// TIA Portal V20 export
FUNCTION_BLOCK "Sequence_10_GaugeRnR"   // FB244, LAD
AUTHOR : ERsystem_FA2_DH. Kim
// stored: IsIECCheckEnabled true, MemoryReserve 100, Namespace Unit1.Em5, SetENOAutomatically false
   VAR_INPUT
      unitStatus : "LAF_typeUnitStatus";
   END_VAR
   VAR
      statSelectedJobNumber { ExternalWritable := 'False'} : DInt;   // Evaluated Job Number
      instSequenceLADStatus { ExternalWritable := 'False'} : "LAF_StatusLadSequence";
      instSequenceLADControl { ExternalWritable := 'False'} : "LAF_ControlLadSequence";
   END_VAR
   VAR CONSTANT
      STEP_IDLE : DInt := 1;
      STEP_IMMEDIATE_STOP : DInt := 9001;   // Step executed when an immediate stop command is triggered for the sequence (i.e. when unit is in state aborting)
      JOB_1_STEP_01 : DInt := 101;
      JOB_1_STEP_10 : DInt := 110;
      JOB_1_STEP_20 : DInt := 120;
      JOB_1_STEP_30 : DInt := 130;
      JOB_1_STEP_90 : DInt := 190;
      JOB_2_STEP_01 : DInt := 201;
      JOB_2_STEP_10 : DInt := 210;
      JOB_2_STEP_20 : DInt := 220;
      JOB_2_STEP_30 : DInt := 230;
      JOB_2_STEP_40 : DInt := 240;
      JOB_2_STEP_50 : DInt := 250;
      JOB_2_STEP_90 : DInt := 290;
      JOB_3_STEP_01 : DInt := 301;
      JOB_3_STEP_10 : DInt := 310;
      JOB_3_STEP_20 : DInt := 320;
      JOB_3_STEP_90 : DInt := 390;
      JOB_4_STEP_01 : DInt := 401;
      JOB_4_STEP_10 : DInt := 410;
      JOB_4_STEP_20 : DInt := 420;
      JOB_4_STEP_30 : DInt := 430;
      JOB_4_STEP_40 : DInt := 440;
      JOB_4_STEP_90 : DInt := 490;
      JOB_5_STEP_01 : DInt := 501;
      JOB_5_STEP_10 : DInt := 510;
      JOB_5_STEP_20 : DInt := 520;
      JOB_5_STEP_90 : DInt := 590;
      JOB_6_STEP_01 : DInt := 601;
      JOB_6_STEP_10 : DInt := 610;
      JOB_6_STEP_20 : DInt := 620;
      JOB_6_STEP_90 : DInt := 690;
      JOB_10_STEP_01 : DInt := 1001;
      JOB_10_STEP_10 : DInt := 1010;
      JOB_10_STEP_20 : DInt := 1020;
      JOB_10_STEP_30 : DInt := 1030;
      JOB_10_STEP_40 : DInt := 1040;
      JOB_10_STEP_90 : DInt := 1090;
      JOB_11_STEP_01 : DInt := 1101;
      JOB_11_STEP_10 : DInt := 1110;
      JOB_11_STEP_20 : DInt := 1120;
      JOB_11_STEP_90 : DInt := 1190;
      JOB_12_STEP_01 : DInt := 1201;
      JOB_12_STEP_10 : DInt := 1210;
      JOB_12_STEP_90 : DInt := 1290;
      JOB_13_STEP_01 : DInt := 1301;
      JOB_13_STEP_10 : DInt := 1310;
      JOB_13_STEP_20 : DInt := 1320;
      JOB_13_STEP_30 : DInt := 1330;
      JOB_13_STEP_40 : DInt := 1340;
      JOB_13_STEP_50 : DInt := 1350;
      JOB_13_STEP_90 : DInt := 1390;
      JOB_15_STEP_01 : DInt := 1501;
      JOB_15_STEP_10 : DInt := 1510;
      JOB_15_STEP_20 : DInt := 1520;
      JOB_15_STEP_90 : DInt := 1590;
      JOB_16_STEP_01 : DInt := 1601;
      JOB_16_STEP_10 : DInt := 1610;
      JOB_16_STEP_20 : DInt := 1620;
      JOB_16_STEP_30 : DInt := 1630;
      JOB_16_STEP_40 : DInt := 1640;
      JOB_16_STEP_90 : DInt := 1690;
      JOB_17_STEP_01 : DInt := 1701;
      JOB_17_STEP_10 : DInt := 1710;
      JOB_17_STEP_20 : DInt := 1720;
      JOB_17_STEP_90 : DInt := 1790;
      JOB_18_STEP_01 : DInt := 1801;
      JOB_18_STEP_10 : DInt := 1810;
      JOB_18_STEP_90 : DInt := 1890;
      JOB_19_STEP_01 : DInt := 1901;
      JOB_19_STEP_10 : DInt := 1910;
      JOB_19_STEP_20 : DInt := 1920;
      JOB_19_STEP_30 : DInt := 1930;
      JOB_19_STEP_40 : DInt := 1940;
      JOB_19_STEP_90 : DInt := 1990;
      JOB_20_STEP_01 : DInt := 2001;
      JOB_20_STEP_10 : DInt := 2010;
      JOB_20_STEP_20 : DInt := 2020;
      JOB_20_STEP_30 : DInt := 2030;
      JOB_20_STEP_40 : DInt := 2040;
      JOB_20_STEP_90 : DInt := 2090;
      JOB_21_STEP_01 : DInt := 2101;
      JOB_21_STEP_10 : DInt := 2110;
      JOB_21_STEP_20 : DInt := 2120;
      JOB_21_STEP_90 : DInt := 2190;
      JOB_22_STEP_01 : DInt := 2201;
      JOB_22_STEP_10 : DInt := 2210;
      JOB_22_STEP_20 : DInt := 2220;
      JOB_22_STEP_30 : DInt := 2230;
      JOB_22_STEP_40 : DInt := 2240;
      JOB_22_STEP_90 : DInt := 2290;
      JOB_23_STEP_01 : DInt := 2301;
      JOB_23_STEP_10 : DInt := 2310;
      JOB_23_STEP_20 : DInt := 2320;
      JOB_23_STEP_90 : DInt := 2390;
      JOB_24_STEP_01 : DInt := 2401;
      JOB_24_STEP_10 : DInt := 2410;
      JOB_24_STEP_20 : DInt := 2420;
      JOB_24_STEP_30 : DInt := 2430;
      JOB_24_STEP_40 : DInt := 2440;
      JOB_24_STEP_90 : DInt := 2490;
      JOB_25_STEP_01 : DInt := 2501;
      JOB_25_STEP_10 : DInt := 2510;
      JOB_25_STEP_20 : DInt := 2520;
      JOB_25_STEP_90 : DInt := 2590;
      JOB_26_STEP_01 : DInt := 2601;
      JOB_26_STEP_10 : DInt := 2610;
      JOB_26_STEP_20 : DInt := 2620;
      JOB_26_STEP_30 : DInt := 2630;
      JOB_26_STEP_40 : DInt := 2640;
      JOB_26_STEP_50 : DInt := 2650;
      JOB_26_STEP_90 : DInt := 2690;
      JOB_30_STEP_01 : DInt := 3001;
      JOB_30_STEP_10 : DInt := 3010;
      JOB_30_STEP_90 : DInt := 3090;
      JOB_31_STEP_01 : DInt := 3101;
      JOB_31_STEP_10 : DInt := 3110;
      JOB_31_STEP_15 : DInt := 3115;
      JOB_31_STEP_20 : DInt := 3120;
      JOB_31_STEP_25 : DInt := 3125;
      JOB_31_STEP_30 : DInt := 3130;
      JOB_31_STEP_35 : DInt := 3135;
      JOB_31_STEP_40 : DInt := 3140;
      JOB_31_STEP_45 : DInt := 3145;
      JOB_31_STEP_50 : DInt := 3150;
      JOB_31_STEP_55 : DInt := 3155;
      JOB_31_STEP_60 : DInt := 3160;
      JOB_31_STEP_65 : DInt := 3165;
      JOB_31_STEP_70 : DInt := 3170;
      JOB_31_STEP_90 : DInt := 3190;
      JOB_32_STEP_01 : DInt := 3201;
      JOB_32_STEP_10 : DInt := 3210;
      JOB_32_STEP_20 : DInt := 3220;
      JOB_32_STEP_90 : DInt := 3290;
      JOB_33_STEP_01 : DInt := 3301;
      JOB_33_STEP_10 : DInt := 3310;
      JOB_33_STEP_90 : DInt := 3390;
      JOB_39_STEP_01 : DInt := 3901;
      JOB_39_STEP_10 : DInt := 3910;
      JOB_39_STEP_90 : DInt := 3990;
   END_VAR
   VAR_TEMP   // added for the SCL form of the ladder/FBD networks
      _w1 : Bool;
   END_VAR
BEGIN

REGION Network 1: BLOCK INFO HEADER
   // (company) / (C) Copyright (year)
   // ---------------------------------------------------------------------------------
   // Title:                             (Title of this block)
   // Comment/Function: (that is implemented in the block)
   // Library/Family:           (that the source is dedicated to)
   // Author:                        (department / person in charge / contact)
   // Target System:          (test system with FW version)
   // Engineering:              TIA Portal (SW version)
   // Restrictions:               (OB types, etc.)
   // Requirements:           (hardware, technological package, etc.)
   // ---------------------------------------------------------------------------------
   // Change log table:
   // Version          | Date             | Signature      | Expert in charge  | Changes applied ------------------------|----------------------|-------------------------|--------------------------------|-----------------------
   // 001.000.000 | yyyy-mm-dd | 0x00000000 | (name of expert) | First released version
END_REGION

REGION Network 2: DESCRIPTION
   // This is a template block provided by the Automation Framework. It can be used to create an own project.
   // The Block Info Header is prepared to put in your own data.
   // Description of the block could be added here and the docu created by Code2Docu.
END_REGION

REGION Network 3: ********************* CONTROL *************************
END_REGION

REGION Network 4: Sequence Control
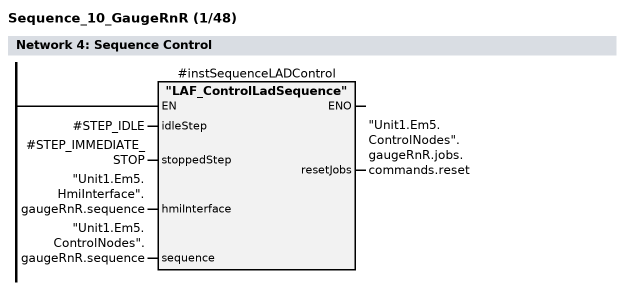
   RUNG wire#powerrail
      #instSequenceLADControl(idleStep := #STEP_IDLE, stoppedStep := #STEP_IMMEDIATE_STOP, hmiInterface := "Unit1.Em5.HmiInterface".gaugeRnR.sequence, sequence := "Unit1.Em5.ControlNodes".gaugeRnR.sequence, resetJobs => "Unit1.Em5.ControlNodes".gaugeRnR.jobs.commands.reset)
   END_RUNG
   // the same network as SCL:
   #instSequenceLADControl(idleStep := #STEP_IDLE,   // "LAF_ControlLadSequence"
                           stoppedStep := #STEP_IMMEDIATE_STOP,
                           hmiInterface := "Unit1.Em5.HmiInterface".gaugeRnR.sequence,
                           sequence := "Unit1.Em5.ControlNodes".gaugeRnR.sequence,
                           resetJobs => "Unit1.Em5.ControlNodes".gaugeRnR.jobs.commands.reset);
END_REGION

REGION Network 5: *************** JOB SELECT **************************
END_REGION

REGION Network 6: STEP IDLE
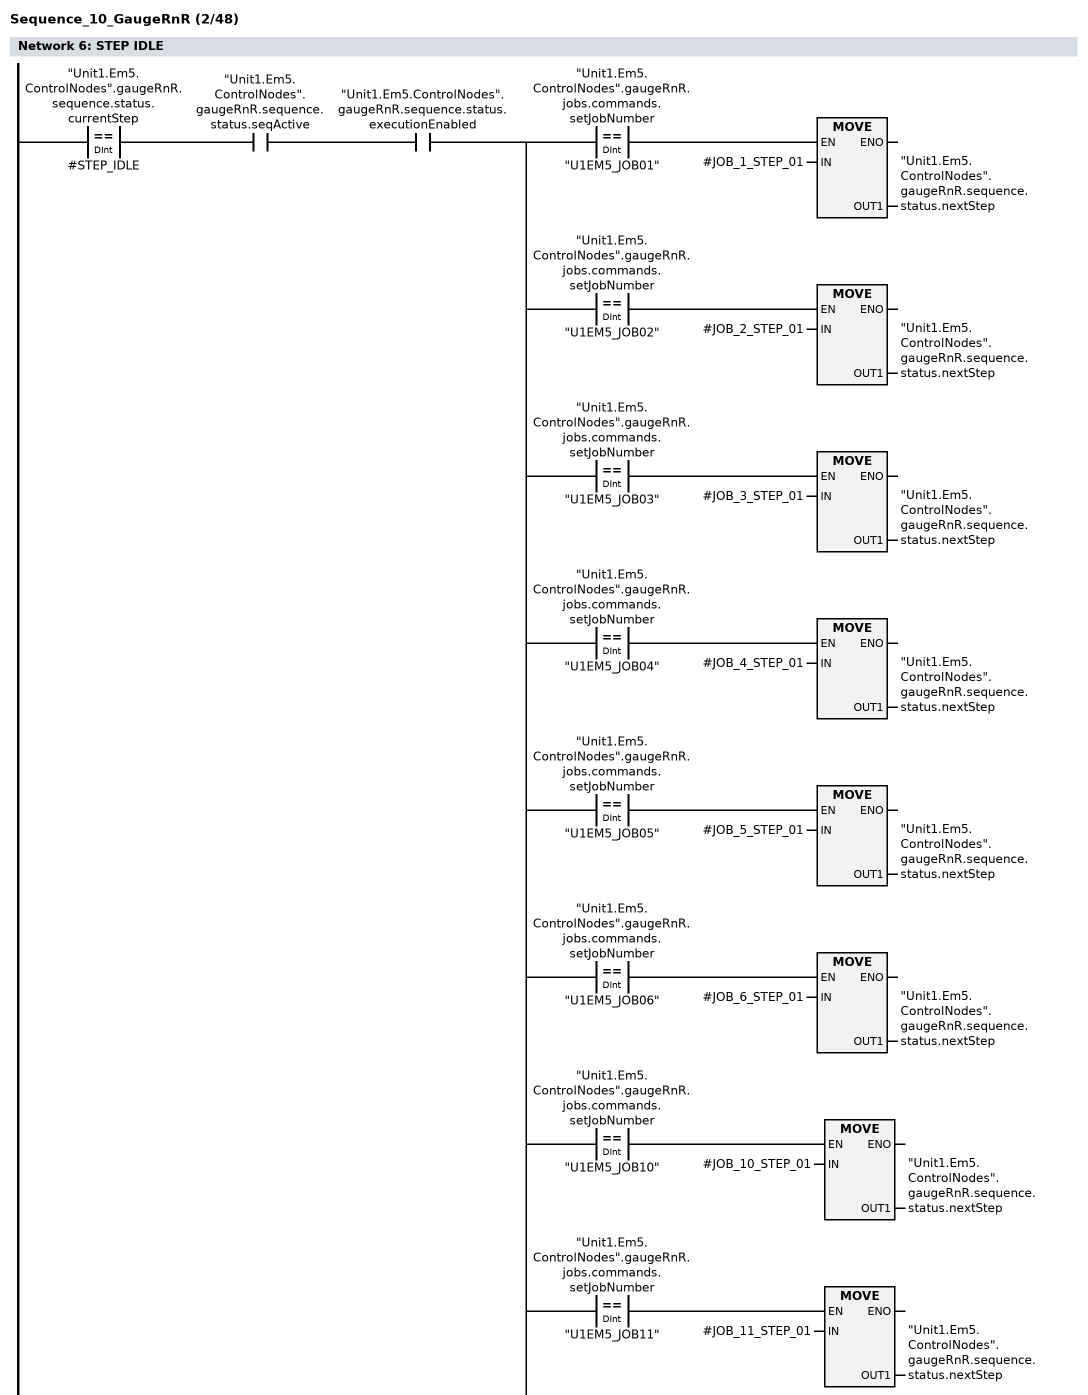
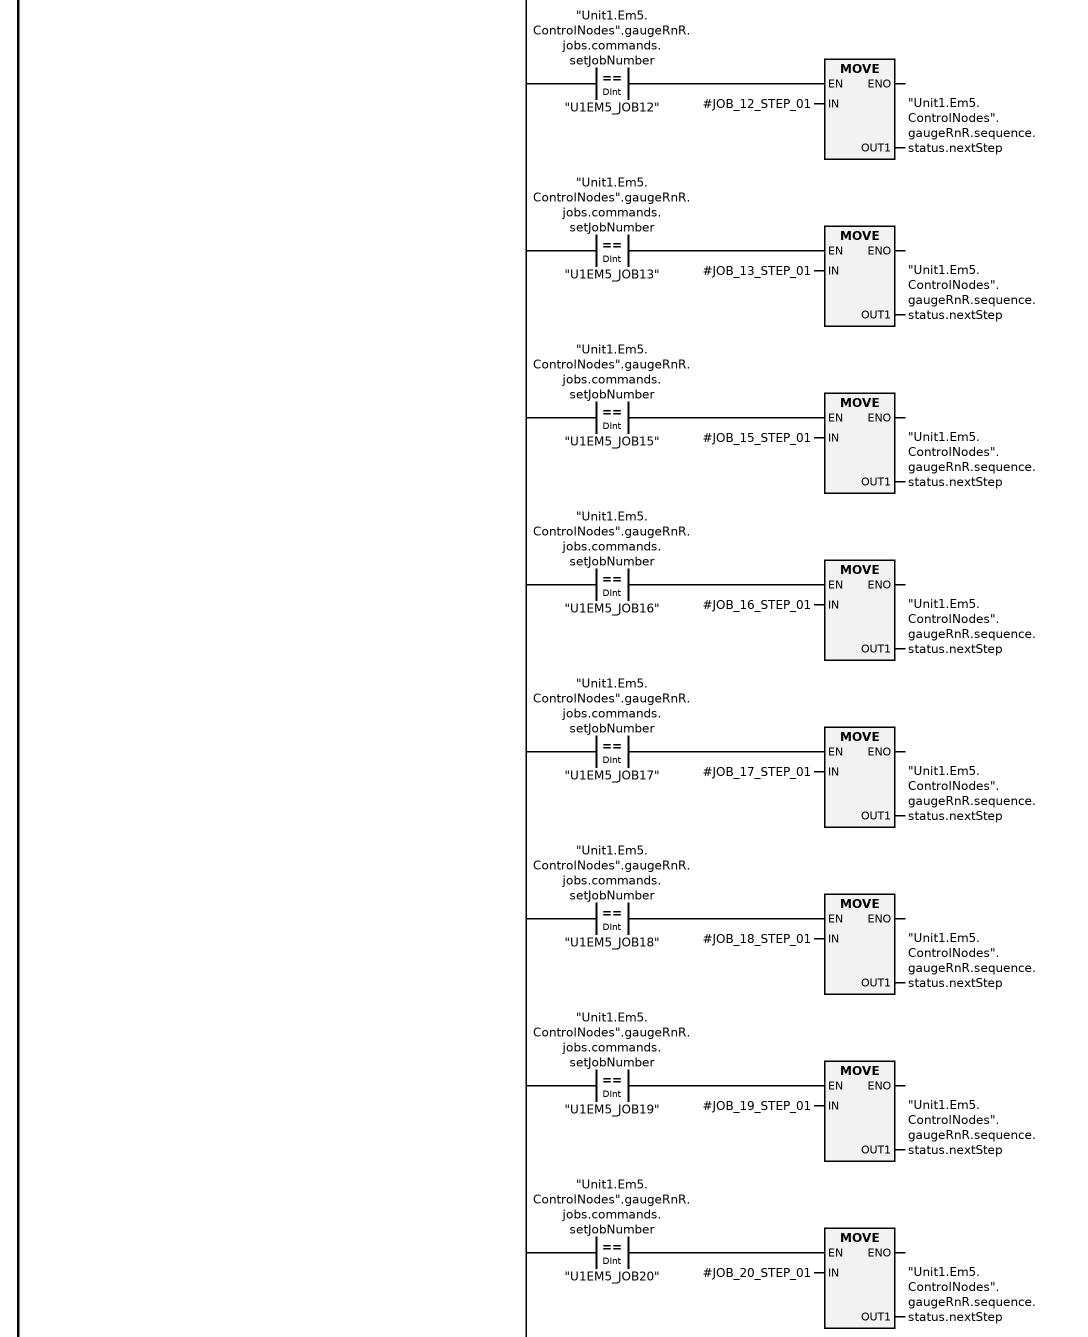
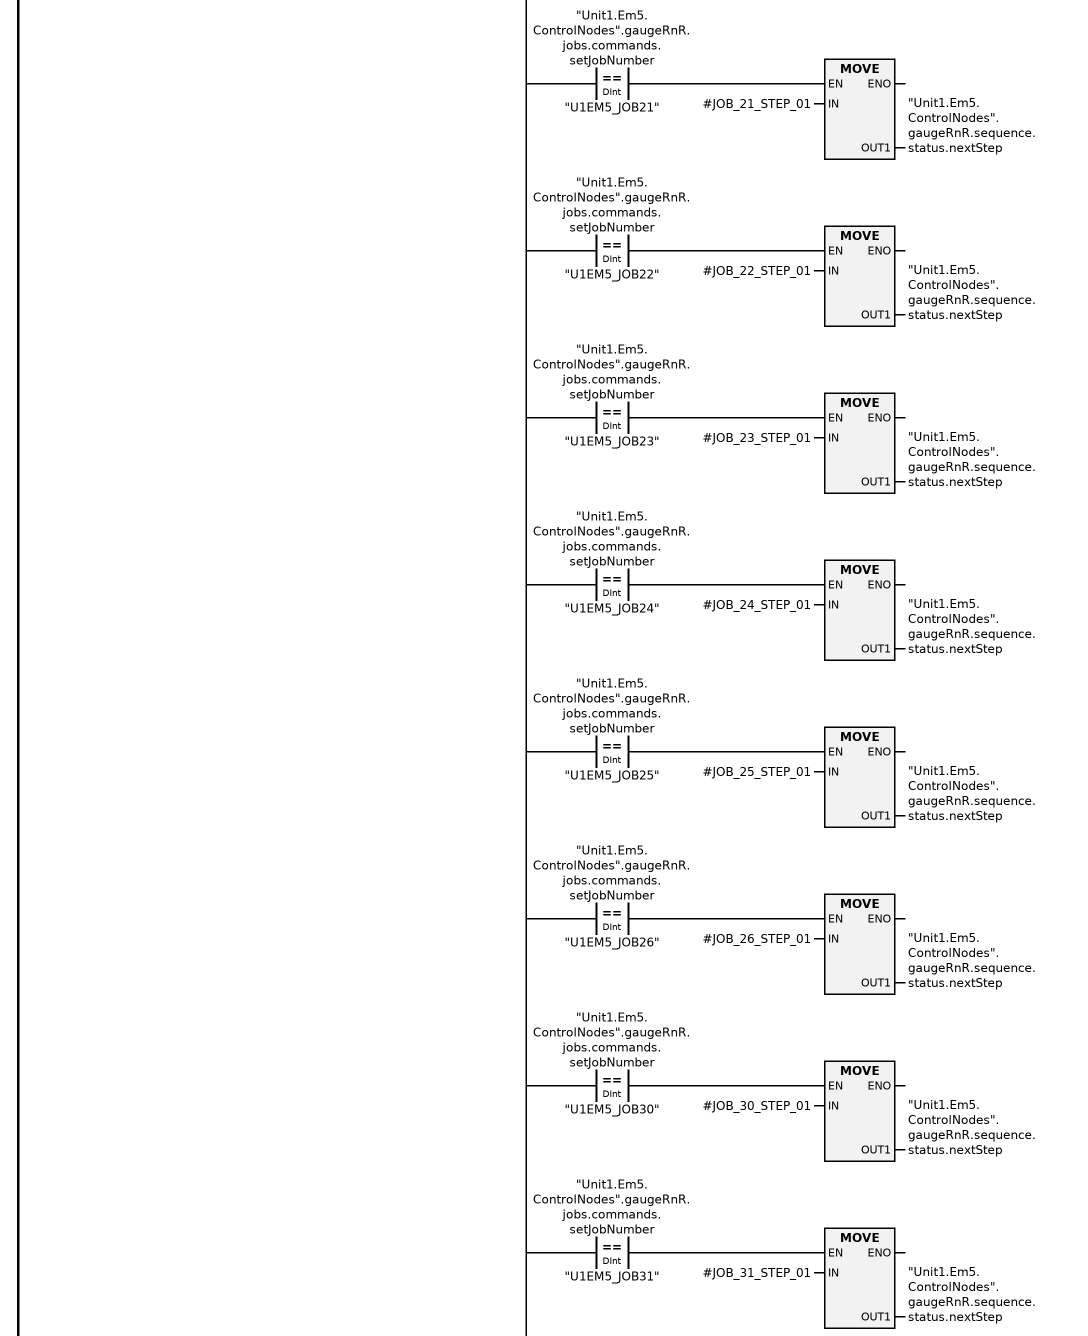
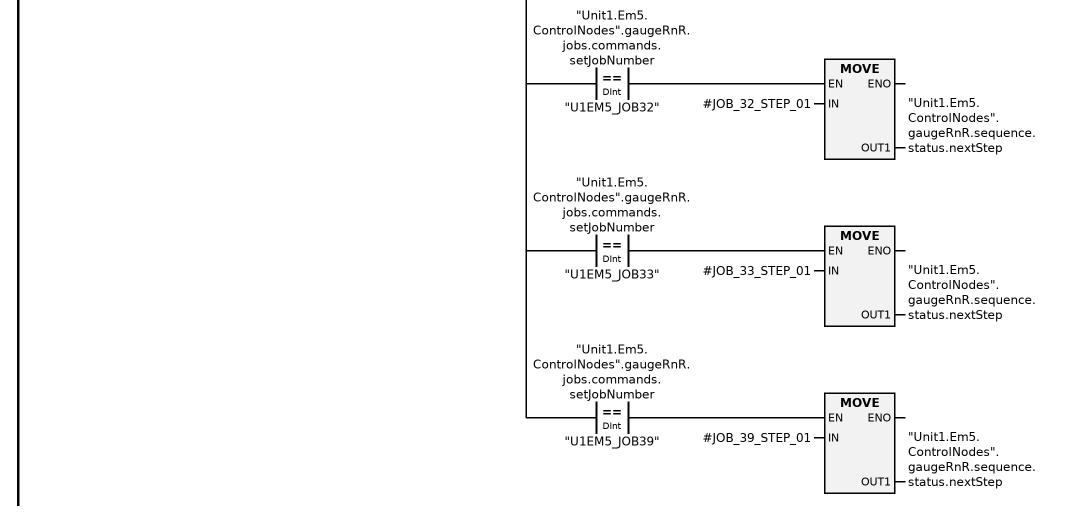
   RUNG wire#powerrail
      { S7_Templates := "SrcType := DInt" } EQ_Contact(in1 := "Unit1.Em5.ControlNodes".gaugeRnR.sequence.status.currentStep, in2 := #STEP_IDLE)
      Contact( "Unit1.Em5.ControlNodes".gaugeRnR.sequence.status.seqActive )
      Contact( "Unit1.Em5.ControlNodes".gaugeRnR.sequence.status.executionEnabled )
      wire#w1
      { S7_Templates := "SrcType := DInt" } EQ_Contact(in1 := "Unit1.Em5.ControlNodes".gaugeRnR.jobs.commands.setJobNumber, in2 := "U1EM5_JOB01")
      Move(in := #JOB_1_STEP_01, out1 => "Unit1.Em5.ControlNodes".gaugeRnR.sequence.status.nextStep)
   END_RUNG
   RUNG wire#w1
      { S7_Templates := "SrcType := DInt" } EQ_Contact(in1 := "Unit1.Em5.ControlNodes".gaugeRnR.jobs.commands.setJobNumber, in2 := "U1EM5_JOB02")
      Move(in := #JOB_2_STEP_01, out1 => "Unit1.Em5.ControlNodes".gaugeRnR.sequence.status.nextStep)
   END_RUNG
   RUNG wire#w1
      { S7_Templates := "SrcType := DInt" } EQ_Contact(in1 := "Unit1.Em5.ControlNodes".gaugeRnR.jobs.commands.setJobNumber, in2 := "U1EM5_JOB03")
      Move(in := #JOB_3_STEP_01, out1 => "Unit1.Em5.ControlNodes".gaugeRnR.sequence.status.nextStep)
   END_RUNG
   RUNG wire#w1
      { S7_Templates := "SrcType := DInt" } EQ_Contact(in1 := "Unit1.Em5.ControlNodes".gaugeRnR.jobs.commands.setJobNumber, in2 := "U1EM5_JOB04")
      Move(in := #JOB_4_STEP_01, out1 => "Unit1.Em5.ControlNodes".gaugeRnR.sequence.status.nextStep)
   END_RUNG
   RUNG wire#w1
      { S7_Templates := "SrcType := DInt" } EQ_Contact(in1 := "Unit1.Em5.ControlNodes".gaugeRnR.jobs.commands.setJobNumber, in2 := "U1EM5_JOB05")
      Move(in := #JOB_5_STEP_01, out1 => "Unit1.Em5.ControlNodes".gaugeRnR.sequence.status.nextStep)
   END_RUNG
   RUNG wire#w1
      { S7_Templates := "SrcType := DInt" } EQ_Contact(in1 := "Unit1.Em5.ControlNodes".gaugeRnR.jobs.commands.setJobNumber, in2 := "U1EM5_JOB06")
      Move(in := #JOB_6_STEP_01, out1 => "Unit1.Em5.ControlNodes".gaugeRnR.sequence.status.nextStep)
   END_RUNG
   RUNG wire#w1
      { S7_Templates := "SrcType := DInt" } EQ_Contact(in1 := "Unit1.Em5.ControlNodes".gaugeRnR.jobs.commands.setJobNumber, in2 := "U1EM5_JOB10")
      Move(in := #JOB_10_STEP_01, out1 => "Unit1.Em5.ControlNodes".gaugeRnR.sequence.status.nextStep)
   END_RUNG
   RUNG wire#w1
      { S7_Templates := "SrcType := DInt" } EQ_Contact(in1 := "Unit1.Em5.ControlNodes".gaugeRnR.jobs.commands.setJobNumber, in2 := "U1EM5_JOB11")
      Move(in := #JOB_11_STEP_01, out1 => "Unit1.Em5.ControlNodes".gaugeRnR.sequence.status.nextStep)
   END_RUNG
   RUNG wire#w1
      { S7_Templates := "SrcType := DInt" } EQ_Contact(in1 := "Unit1.Em5.ControlNodes".gaugeRnR.jobs.commands.setJobNumber, in2 := "U1EM5_JOB12")
      Move(in := #JOB_12_STEP_01, out1 => "Unit1.Em5.ControlNodes".gaugeRnR.sequence.status.nextStep)
   END_RUNG
   RUNG wire#w1
      { S7_Templates := "SrcType := DInt" } EQ_Contact(in1 := "Unit1.Em5.ControlNodes".gaugeRnR.jobs.commands.setJobNumber, in2 := "U1EM5_JOB13")
      Move(in := #JOB_13_STEP_01, out1 => "Unit1.Em5.ControlNodes".gaugeRnR.sequence.status.nextStep)
   END_RUNG
   RUNG wire#w1
      { S7_Templates := "SrcType := DInt" } EQ_Contact(in1 := "Unit1.Em5.ControlNodes".gaugeRnR.jobs.commands.setJobNumber, in2 := "U1EM5_JOB15")
      Move(in := #JOB_15_STEP_01, out1 => "Unit1.Em5.ControlNodes".gaugeRnR.sequence.status.nextStep)
   END_RUNG
   RUNG wire#w1
      { S7_Templates := "SrcType := DInt" } EQ_Contact(in1 := "Unit1.Em5.ControlNodes".gaugeRnR.jobs.commands.setJobNumber, in2 := "U1EM5_JOB16")
      Move(in := #JOB_16_STEP_01, out1 => "Unit1.Em5.ControlNodes".gaugeRnR.sequence.status.nextStep)
   END_RUNG
   RUNG wire#w1
      { S7_Templates := "SrcType := DInt" } EQ_Contact(in1 := "Unit1.Em5.ControlNodes".gaugeRnR.jobs.commands.setJobNumber, in2 := "U1EM5_JOB17")
      Move(in := #JOB_17_STEP_01, out1 => "Unit1.Em5.ControlNodes".gaugeRnR.sequence.status.nextStep)
   END_RUNG
   RUNG wire#w1
      { S7_Templates := "SrcType := DInt" } EQ_Contact(in1 := "Unit1.Em5.ControlNodes".gaugeRnR.jobs.commands.setJobNumber, in2 := "U1EM5_JOB18")
      Move(in := #JOB_18_STEP_01, out1 => "Unit1.Em5.ControlNodes".gaugeRnR.sequence.status.nextStep)
   END_RUNG
   RUNG wire#w1
      { S7_Templates := "SrcType := DInt" } EQ_Contact(in1 := "Unit1.Em5.ControlNodes".gaugeRnR.jobs.commands.setJobNumber, in2 := "U1EM5_JOB19")
      Move(in := #JOB_19_STEP_01, out1 => "Unit1.Em5.ControlNodes".gaugeRnR.sequence.status.nextStep)
   END_RUNG
   RUNG wire#w1
      { S7_Templates := "SrcType := DInt" } EQ_Contact(in1 := "Unit1.Em5.ControlNodes".gaugeRnR.jobs.commands.setJobNumber, in2 := "U1EM5_JOB20")
      Move(in := #JOB_20_STEP_01, out1 => "Unit1.Em5.ControlNodes".gaugeRnR.sequence.status.nextStep)
   END_RUNG
   RUNG wire#w1
      { S7_Templates := "SrcType := DInt" } EQ_Contact(in1 := "Unit1.Em5.ControlNodes".gaugeRnR.jobs.commands.setJobNumber, in2 := "U1EM5_JOB21")
      Move(in := #JOB_21_STEP_01, out1 => "Unit1.Em5.ControlNodes".gaugeRnR.sequence.status.nextStep)
   END_RUNG
   RUNG wire#w1
      { S7_Templates := "SrcType := DInt" } EQ_Contact(in1 := "Unit1.Em5.ControlNodes".gaugeRnR.jobs.commands.setJobNumber, in2 := "U1EM5_JOB22")
      Move(in := #JOB_22_STEP_01, out1 => "Unit1.Em5.ControlNodes".gaugeRnR.sequence.status.nextStep)
   END_RUNG
   RUNG wire#w1
      { S7_Templates := "SrcType := DInt" } EQ_Contact(in1 := "Unit1.Em5.ControlNodes".gaugeRnR.jobs.commands.setJobNumber, in2 := "U1EM5_JOB23")
      Move(in := #JOB_23_STEP_01, out1 => "Unit1.Em5.ControlNodes".gaugeRnR.sequence.status.nextStep)
   END_RUNG
   RUNG wire#w1
      { S7_Templates := "SrcType := DInt" } EQ_Contact(in1 := "Unit1.Em5.ControlNodes".gaugeRnR.jobs.commands.setJobNumber, in2 := "U1EM5_JOB24")
      Move(in := #JOB_24_STEP_01, out1 => "Unit1.Em5.ControlNodes".gaugeRnR.sequence.status.nextStep)
   END_RUNG
   RUNG wire#w1
      { S7_Templates := "SrcType := DInt" } EQ_Contact(in1 := "Unit1.Em5.ControlNodes".gaugeRnR.jobs.commands.setJobNumber, in2 := "U1EM5_JOB25")
      Move(in := #JOB_25_STEP_01, out1 => "Unit1.Em5.ControlNodes".gaugeRnR.sequence.status.nextStep)
   END_RUNG
   RUNG wire#w1
      { S7_Templates := "SrcType := DInt" } EQ_Contact(in1 := "Unit1.Em5.ControlNodes".gaugeRnR.jobs.commands.setJobNumber, in2 := "U1EM5_JOB26")
      Move(in := #JOB_26_STEP_01, out1 => "Unit1.Em5.ControlNodes".gaugeRnR.sequence.status.nextStep)
   END_RUNG
   RUNG wire#w1
      { S7_Templates := "SrcType := DInt" } EQ_Contact(in1 := "Unit1.Em5.ControlNodes".gaugeRnR.jobs.commands.setJobNumber, in2 := "U1EM5_JOB30")
      Move(in := #JOB_30_STEP_01, out1 => "Unit1.Em5.ControlNodes".gaugeRnR.sequence.status.nextStep)
   END_RUNG
   RUNG wire#w1
      { S7_Templates := "SrcType := DInt" } EQ_Contact(in1 := "Unit1.Em5.ControlNodes".gaugeRnR.jobs.commands.setJobNumber, in2 := "U1EM5_JOB31")
      Move(in := #JOB_31_STEP_01, out1 => "Unit1.Em5.ControlNodes".gaugeRnR.sequence.status.nextStep)
   END_RUNG
   RUNG wire#w1
      { S7_Templates := "SrcType := DInt" } EQ_Contact(in1 := "Unit1.Em5.ControlNodes".gaugeRnR.jobs.commands.setJobNumber, in2 := "U1EM5_JOB32")
      Move(in := #JOB_32_STEP_01, out1 => "Unit1.Em5.ControlNodes".gaugeRnR.sequence.status.nextStep)
   END_RUNG
   RUNG wire#w1
      { S7_Templates := "SrcType := DInt" } EQ_Contact(in1 := "Unit1.Em5.ControlNodes".gaugeRnR.jobs.commands.setJobNumber, in2 := "U1EM5_JOB33")
      Move(in := #JOB_33_STEP_01, out1 => "Unit1.Em5.ControlNodes".gaugeRnR.sequence.status.nextStep)
   END_RUNG
   RUNG wire#w1
      { S7_Templates := "SrcType := DInt" } EQ_Contact(in1 := "Unit1.Em5.ControlNodes".gaugeRnR.jobs.commands.setJobNumber, in2 := "U1EM5_JOB39")
      Move(in := #JOB_39_STEP_01, out1 => "Unit1.Em5.ControlNodes".gaugeRnR.sequence.status.nextStep)
   END_RUNG
   // the same network as SCL:
   #_w1 := ("Unit1.Em5.ControlNodes".gaugeRnR.sequence.status.currentStep = #STEP_IDLE) AND "Unit1.Em5.ControlNodes".gaugeRnR.sequence.status.seqActive AND "Unit1.Em5.ControlNodes".gaugeRnR.sequence.status.executionEnabled;
   IF #_w1 AND ("Unit1.Em5.ControlNodes".gaugeRnR.jobs.commands.setJobNumber = "U1EM5_JOB01") THEN
       "Unit1.Em5.ControlNodes".gaugeRnR.sequence.status.nextStep := #JOB_1_STEP_01;
   END_IF;
   IF #_w1 AND ("Unit1.Em5.ControlNodes".gaugeRnR.jobs.commands.setJobNumber = "U1EM5_JOB02") THEN
       "Unit1.Em5.ControlNodes".gaugeRnR.sequence.status.nextStep := #JOB_2_STEP_01;
   END_IF;
   IF #_w1 AND ("Unit1.Em5.ControlNodes".gaugeRnR.jobs.commands.setJobNumber = "U1EM5_JOB03") THEN
       "Unit1.Em5.ControlNodes".gaugeRnR.sequence.status.nextStep := #JOB_3_STEP_01;
   END_IF;
   IF #_w1 AND ("Unit1.Em5.ControlNodes".gaugeRnR.jobs.commands.setJobNumber = "U1EM5_JOB04") THEN
       "Unit1.Em5.ControlNodes".gaugeRnR.sequence.status.nextStep := #JOB_4_STEP_01;
   END_IF;
   IF #_w1 AND ("Unit1.Em5.ControlNodes".gaugeRnR.jobs.commands.setJobNumber = "U1EM5_JOB05") THEN
       "Unit1.Em5.ControlNodes".gaugeRnR.sequence.status.nextStep := #JOB_5_STEP_01;
   END_IF;
   IF #_w1 AND ("Unit1.Em5.ControlNodes".gaugeRnR.jobs.commands.setJobNumber = "U1EM5_JOB06") THEN
       "Unit1.Em5.ControlNodes".gaugeRnR.sequence.status.nextStep := #JOB_6_STEP_01;
   END_IF;
   IF #_w1 AND ("Unit1.Em5.ControlNodes".gaugeRnR.jobs.commands.setJobNumber = "U1EM5_JOB10") THEN
       "Unit1.Em5.ControlNodes".gaugeRnR.sequence.status.nextStep := #JOB_10_STEP_01;
   END_IF;
   IF #_w1 AND ("Unit1.Em5.ControlNodes".gaugeRnR.jobs.commands.setJobNumber = "U1EM5_JOB11") THEN
       "Unit1.Em5.ControlNodes".gaugeRnR.sequence.status.nextStep := #JOB_11_STEP_01;
   END_IF;
   IF #_w1 AND ("Unit1.Em5.ControlNodes".gaugeRnR.jobs.commands.setJobNumber = "U1EM5_JOB12") THEN
       "Unit1.Em5.ControlNodes".gaugeRnR.sequence.status.nextStep := #JOB_12_STEP_01;
   END_IF;
   IF #_w1 AND ("Unit1.Em5.ControlNodes".gaugeRnR.jobs.commands.setJobNumber = "U1EM5_JOB13") THEN
       "Unit1.Em5.ControlNodes".gaugeRnR.sequence.status.nextStep := #JOB_13_STEP_01;
   END_IF;
   IF #_w1 AND ("Unit1.Em5.ControlNodes".gaugeRnR.jobs.commands.setJobNumber = "U1EM5_JOB15") THEN
       "Unit1.Em5.ControlNodes".gaugeRnR.sequence.status.nextStep := #JOB_15_STEP_01;
   END_IF;
   IF #_w1 AND ("Unit1.Em5.ControlNodes".gaugeRnR.jobs.commands.setJobNumber = "U1EM5_JOB16") THEN
       "Unit1.Em5.ControlNodes".gaugeRnR.sequence.status.nextStep := #JOB_16_STEP_01;
   END_IF;
   IF #_w1 AND ("Unit1.Em5.ControlNodes".gaugeRnR.jobs.commands.setJobNumber = "U1EM5_JOB17") THEN
       "Unit1.Em5.ControlNodes".gaugeRnR.sequence.status.nextStep := #JOB_17_STEP_01;
   END_IF;
   IF #_w1 AND ("Unit1.Em5.ControlNodes".gaugeRnR.jobs.commands.setJobNumber = "U1EM5_JOB18") THEN
       "Unit1.Em5.ControlNodes".gaugeRnR.sequence.status.nextStep := #JOB_18_STEP_01;
   END_IF;
   IF #_w1 AND ("Unit1.Em5.ControlNodes".gaugeRnR.jobs.commands.setJobNumber = "U1EM5_JOB19") THEN
       "Unit1.Em5.ControlNodes".gaugeRnR.sequence.status.nextStep := #JOB_19_STEP_01;
   END_IF;
   IF #_w1 AND ("Unit1.Em5.ControlNodes".gaugeRnR.jobs.commands.setJobNumber = "U1EM5_JOB20") THEN
       "Unit1.Em5.ControlNodes".gaugeRnR.sequence.status.nextStep := #JOB_20_STEP_01;
   END_IF;
   IF #_w1 AND ("Unit1.Em5.ControlNodes".gaugeRnR.jobs.commands.setJobNumber = "U1EM5_JOB21") THEN
       "Unit1.Em5.ControlNodes".gaugeRnR.sequence.status.nextStep := #JOB_21_STEP_01;
   END_IF;
   IF #_w1 AND ("Unit1.Em5.ControlNodes".gaugeRnR.jobs.commands.setJobNumber = "U1EM5_JOB22") THEN
       "Unit1.Em5.ControlNodes".gaugeRnR.sequence.status.nextStep := #JOB_22_STEP_01;
   END_IF;
   IF #_w1 AND ("Unit1.Em5.ControlNodes".gaugeRnR.jobs.commands.setJobNumber = "U1EM5_JOB23") THEN
       "Unit1.Em5.ControlNodes".gaugeRnR.sequence.status.nextStep := #JOB_23_STEP_01;
   END_IF;
   IF #_w1 AND ("Unit1.Em5.ControlNodes".gaugeRnR.jobs.commands.setJobNumber = "U1EM5_JOB24") THEN
       "Unit1.Em5.ControlNodes".gaugeRnR.sequence.status.nextStep := #JOB_24_STEP_01;
   END_IF;
   IF #_w1 AND ("Unit1.Em5.ControlNodes".gaugeRnR.jobs.commands.setJobNumber = "U1EM5_JOB25") THEN
       "Unit1.Em5.ControlNodes".gaugeRnR.sequence.status.nextStep := #JOB_25_STEP_01;
   END_IF;
   IF #_w1 AND ("Unit1.Em5.ControlNodes".gaugeRnR.jobs.commands.setJobNumber = "U1EM5_JOB26") THEN
       "Unit1.Em5.ControlNodes".gaugeRnR.sequence.status.nextStep := #JOB_26_STEP_01;
   END_IF;
   IF #_w1 AND ("Unit1.Em5.ControlNodes".gaugeRnR.jobs.commands.setJobNumber = "U1EM5_JOB30") THEN
       "Unit1.Em5.ControlNodes".gaugeRnR.sequence.status.nextStep := #JOB_30_STEP_01;
   END_IF;
   IF #_w1 AND ("Unit1.Em5.ControlNodes".gaugeRnR.jobs.commands.setJobNumber = "U1EM5_JOB31") THEN
       "Unit1.Em5.ControlNodes".gaugeRnR.sequence.status.nextStep := #JOB_31_STEP_01;
   END_IF;
   IF #_w1 AND ("Unit1.Em5.ControlNodes".gaugeRnR.jobs.commands.setJobNumber = "U1EM5_JOB32") THEN
       "Unit1.Em5.ControlNodes".gaugeRnR.sequence.status.nextStep := #JOB_32_STEP_01;
   END_IF;
   IF #_w1 AND ("Unit1.Em5.ControlNodes".gaugeRnR.jobs.commands.setJobNumber = "U1EM5_JOB33") THEN
       "Unit1.Em5.ControlNodes".gaugeRnR.sequence.status.nextStep := #JOB_33_STEP_01;
   END_IF;
   IF #_w1 AND ("Unit1.Em5.ControlNodes".gaugeRnR.jobs.commands.setJobNumber = "U1EM5_JOB39") THEN
       "Unit1.Em5.ControlNodes".gaugeRnR.sequence.status.nextStep := #JOB_39_STEP_01;
   END_IF;
END_REGION

REGION Network 7: *************** JOB[1] Common GugeRnR Ready ************************
END_REGION

REGION Network 8: Step[101] : JOB[1] Condition
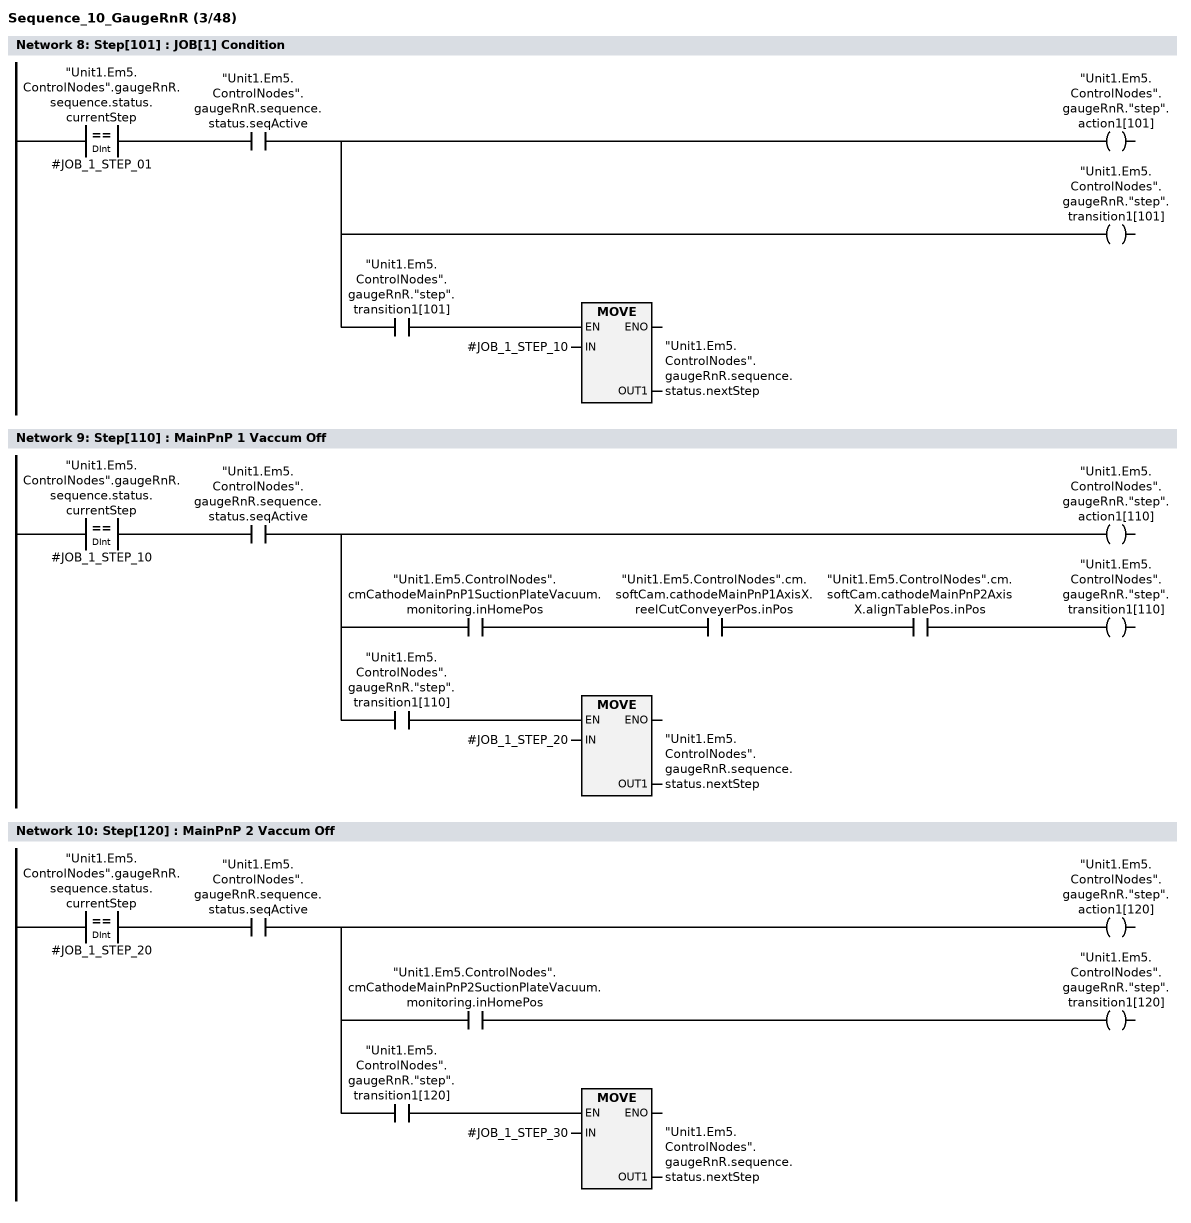
   RUNG wire#powerrail
      { S7_Templates := "SrcType := DInt" } EQ_Contact(in1 := "Unit1.Em5.ControlNodes".gaugeRnR.sequence.status.currentStep, in2 := #JOB_1_STEP_01)
      Contact( "Unit1.Em5.ControlNodes".gaugeRnR.sequence.status.seqActive )
      wire#w1
      Coil( "Unit1.Em5.ControlNodes".gaugeRnR."step".action1[101] )
   END_RUNG
   RUNG wire#w1
      Coil( "Unit1.Em5.ControlNodes".gaugeRnR."step".transition1[101] )
   END_RUNG
   RUNG wire#w1
      Contact( "Unit1.Em5.ControlNodes".gaugeRnR."step".transition1[101] )
      Move(in := #JOB_1_STEP_10, out1 => "Unit1.Em5.ControlNodes".gaugeRnR.sequence.status.nextStep)
   END_RUNG
   // the same network as SCL:
   "Unit1.Em5.ControlNodes".gaugeRnR."step".action1[101] := ("Unit1.Em5.ControlNodes".gaugeRnR.sequence.status.currentStep = #JOB_1_STEP_01) AND "Unit1.Em5.ControlNodes".gaugeRnR.sequence.status.seqActive;
   "Unit1.Em5.ControlNodes".gaugeRnR."step".transition1[101] := ("Unit1.Em5.ControlNodes".gaugeRnR.sequence.status.currentStep = #JOB_1_STEP_01) AND "Unit1.Em5.ControlNodes".gaugeRnR.sequence.status.seqActive;
   IF ("Unit1.Em5.ControlNodes".gaugeRnR.sequence.status.currentStep = #JOB_1_STEP_01) AND "Unit1.Em5.ControlNodes".gaugeRnR.sequence.status.seqActive AND "Unit1.Em5.ControlNodes".gaugeRnR."step".transition1[101] THEN
       "Unit1.Em5.ControlNodes".gaugeRnR.sequence.status.nextStep := #JOB_1_STEP_10;
   END_IF;
END_REGION

REGION Network 9: Step[110] : MainPnP 1 Vaccum Off
   RUNG wire#powerrail
      { S7_Templates := "SrcType := DInt" } EQ_Contact(in1 := "Unit1.Em5.ControlNodes".gaugeRnR.sequence.status.currentStep, in2 := #JOB_1_STEP_10)
      Contact( "Unit1.Em5.ControlNodes".gaugeRnR.sequence.status.seqActive )
      wire#w1
      Coil( "Unit1.Em5.ControlNodes".gaugeRnR."step".action1[110] )
   END_RUNG
   RUNG wire#w1
      Contact( "Unit1.Em5.ControlNodes".cmCathodeMainPnP1SuctionPlateVacuum.monitoring.inHomePos )
      Contact( "Unit1.Em5.ControlNodes".cm.softCam.cathodeMainPnP1AxisX.reelCutConveyerPos.inPos )
      Contact( "Unit1.Em5.ControlNodes".cm.softCam.cathodeMainPnP2AxisX.alignTablePos.inPos )
      Coil( "Unit1.Em5.ControlNodes".gaugeRnR."step".transition1[110] )
   END_RUNG
   RUNG wire#w1
      Contact( "Unit1.Em5.ControlNodes".gaugeRnR."step".transition1[110] )
      Move(in := #JOB_1_STEP_20, out1 => "Unit1.Em5.ControlNodes".gaugeRnR.sequence.status.nextStep)
   END_RUNG
   // the same network as SCL:
   "Unit1.Em5.ControlNodes".gaugeRnR."step".action1[110] := ("Unit1.Em5.ControlNodes".gaugeRnR.sequence.status.currentStep = #JOB_1_STEP_10) AND "Unit1.Em5.ControlNodes".gaugeRnR.sequence.status.seqActive;
   "Unit1.Em5.ControlNodes".gaugeRnR."step".transition1[110] := ("Unit1.Em5.ControlNodes".gaugeRnR.sequence.status.currentStep = #JOB_1_STEP_10) AND "Unit1.Em5.ControlNodes".gaugeRnR.sequence.status.seqActive AND "Unit1.Em5.ControlNodes".cmCathodeMainPnP1SuctionPlateVacuum.monitoring.inHomePos AND "Unit1.Em5.ControlNodes".cm.softCam.cathodeMainPnP1AxisX.reelCutConveyerPos.inPos AND "Unit1.Em5.ControlNodes".cm.softCam.cathodeMainPnP2AxisX.alignTablePos.inPos;
   IF ("Unit1.Em5.ControlNodes".gaugeRnR.sequence.status.currentStep = #JOB_1_STEP_10) AND "Unit1.Em5.ControlNodes".gaugeRnR.sequence.status.seqActive AND "Unit1.Em5.ControlNodes".gaugeRnR."step".transition1[110] THEN
       "Unit1.Em5.ControlNodes".gaugeRnR.sequence.status.nextStep := #JOB_1_STEP_20;
   END_IF;
END_REGION

REGION Network 10: Step[120] : MainPnP 2 Vaccum Off
   RUNG wire#powerrail
      { S7_Templates := "SrcType := DInt" } EQ_Contact(in1 := "Unit1.Em5.ControlNodes".gaugeRnR.sequence.status.currentStep, in2 := #JOB_1_STEP_20)
      Contact( "Unit1.Em5.ControlNodes".gaugeRnR.sequence.status.seqActive )
      wire#w1
      Coil( "Unit1.Em5.ControlNodes".gaugeRnR."step".action1[120] )
   END_RUNG
   RUNG wire#w1
      Contact( "Unit1.Em5.ControlNodes".cmCathodeMainPnP2SuctionPlateVacuum.monitoring.inHomePos )
      Coil( "Unit1.Em5.ControlNodes".gaugeRnR."step".transition1[120] )
   END_RUNG
   RUNG wire#w1
      Contact( "Unit1.Em5.ControlNodes".gaugeRnR."step".transition1[120] )
      Move(in := #JOB_1_STEP_30, out1 => "Unit1.Em5.ControlNodes".gaugeRnR.sequence.status.nextStep)
   END_RUNG
   // the same network as SCL:
   "Unit1.Em5.ControlNodes".gaugeRnR."step".action1[120] := ("Unit1.Em5.ControlNodes".gaugeRnR.sequence.status.currentStep = #JOB_1_STEP_20) AND "Unit1.Em5.ControlNodes".gaugeRnR.sequence.status.seqActive;
   "Unit1.Em5.ControlNodes".gaugeRnR."step".transition1[120] := ("Unit1.Em5.ControlNodes".gaugeRnR.sequence.status.currentStep = #JOB_1_STEP_20) AND "Unit1.Em5.ControlNodes".gaugeRnR.sequence.status.seqActive AND "Unit1.Em5.ControlNodes".cmCathodeMainPnP2SuctionPlateVacuum.monitoring.inHomePos;
   IF ("Unit1.Em5.ControlNodes".gaugeRnR.sequence.status.currentStep = #JOB_1_STEP_20) AND "Unit1.Em5.ControlNodes".gaugeRnR.sequence.status.seqActive AND "Unit1.Em5.ControlNodes".gaugeRnR."step".transition1[120] THEN
       "Unit1.Em5.ControlNodes".gaugeRnR.sequence.status.nextStep := #JOB_1_STEP_30;
   END_IF;
END_REGION

REGION Network 11: Step[130] : AlignTable Vaccum Off
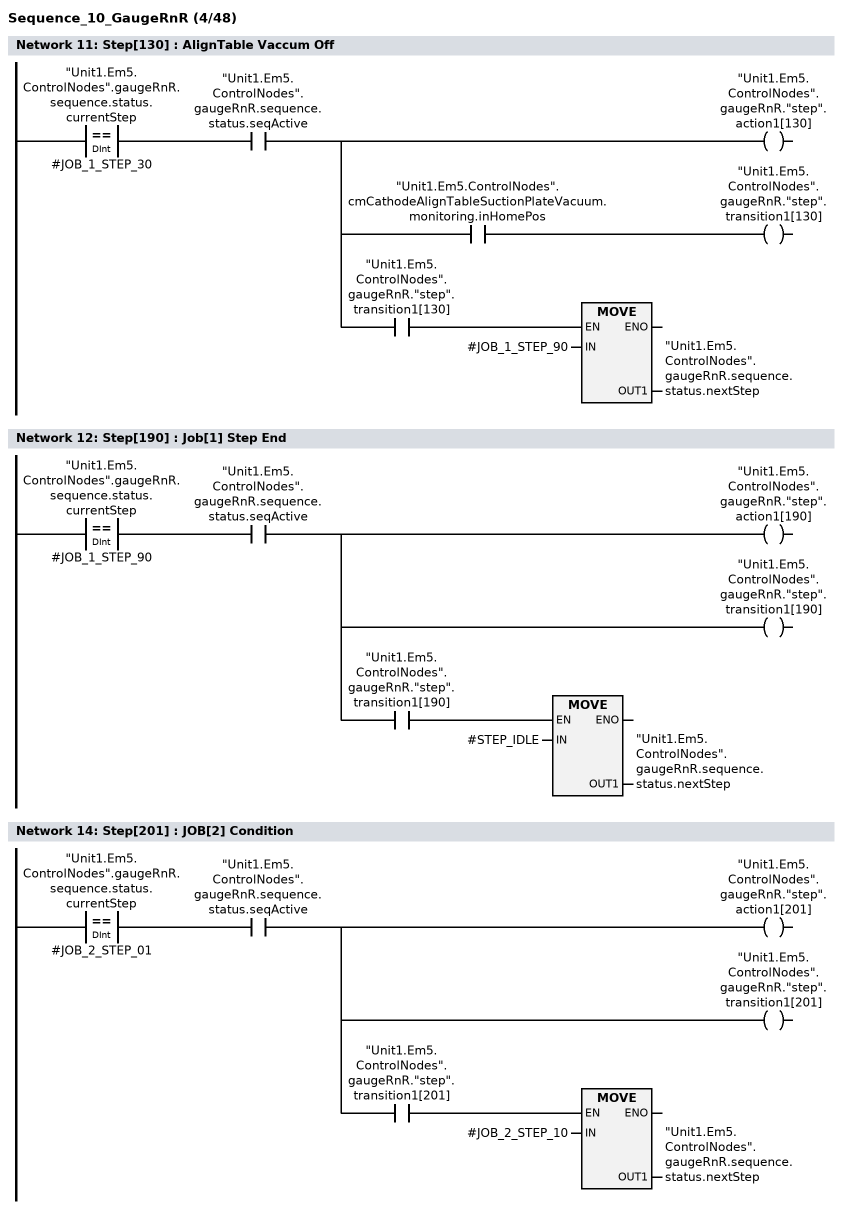
   RUNG wire#powerrail
      { S7_Templates := "SrcType := DInt" } EQ_Contact(in1 := "Unit1.Em5.ControlNodes".gaugeRnR.sequence.status.currentStep, in2 := #JOB_1_STEP_30)
      Contact( "Unit1.Em5.ControlNodes".gaugeRnR.sequence.status.seqActive )
      wire#w1
      Coil( "Unit1.Em5.ControlNodes".gaugeRnR."step".action1[130] )
   END_RUNG
   RUNG wire#w1
      Contact( "Unit1.Em5.ControlNodes".cmCathodeAlignTableSuctionPlateVacuum.monitoring.inHomePos )
      Coil( "Unit1.Em5.ControlNodes".gaugeRnR."step".transition1[130] )
   END_RUNG
   RUNG wire#w1
      Contact( "Unit1.Em5.ControlNodes".gaugeRnR."step".transition1[130] )
      Move(in := #JOB_1_STEP_90, out1 => "Unit1.Em5.ControlNodes".gaugeRnR.sequence.status.nextStep)
   END_RUNG
   // the same network as SCL:
   "Unit1.Em5.ControlNodes".gaugeRnR."step".action1[130] := ("Unit1.Em5.ControlNodes".gaugeRnR.sequence.status.currentStep = #JOB_1_STEP_30) AND "Unit1.Em5.ControlNodes".gaugeRnR.sequence.status.seqActive;
   "Unit1.Em5.ControlNodes".gaugeRnR."step".transition1[130] := ("Unit1.Em5.ControlNodes".gaugeRnR.sequence.status.currentStep = #JOB_1_STEP_30) AND "Unit1.Em5.ControlNodes".gaugeRnR.sequence.status.seqActive AND "Unit1.Em5.ControlNodes".cmCathodeAlignTableSuctionPlateVacuum.monitoring.inHomePos;
   IF ("Unit1.Em5.ControlNodes".gaugeRnR.sequence.status.currentStep = #JOB_1_STEP_30) AND "Unit1.Em5.ControlNodes".gaugeRnR.sequence.status.seqActive AND "Unit1.Em5.ControlNodes".gaugeRnR."step".transition1[130] THEN
       "Unit1.Em5.ControlNodes".gaugeRnR.sequence.status.nextStep := #JOB_1_STEP_90;
   END_IF;
END_REGION

REGION Network 12: Step[190] : Job[1] Step End
   RUNG wire#powerrail
      { S7_Templates := "SrcType := DInt" } EQ_Contact(in1 := "Unit1.Em5.ControlNodes".gaugeRnR.sequence.status.currentStep, in2 := #JOB_1_STEP_90)
      Contact( "Unit1.Em5.ControlNodes".gaugeRnR.sequence.status.seqActive )
      wire#w1
      Coil( "Unit1.Em5.ControlNodes".gaugeRnR."step".action1[190] )
   END_RUNG
   RUNG wire#w1
      Coil( "Unit1.Em5.ControlNodes".gaugeRnR."step".transition1[190] )
   END_RUNG
   RUNG wire#w1
      Contact( "Unit1.Em5.ControlNodes".gaugeRnR."step".transition1[190] )
      Move(in := #STEP_IDLE, out1 => "Unit1.Em5.ControlNodes".gaugeRnR.sequence.status.nextStep)
   END_RUNG
   // the same network as SCL:
   "Unit1.Em5.ControlNodes".gaugeRnR."step".action1[190] := ("Unit1.Em5.ControlNodes".gaugeRnR.sequence.status.currentStep = #JOB_1_STEP_90) AND "Unit1.Em5.ControlNodes".gaugeRnR.sequence.status.seqActive;
   "Unit1.Em5.ControlNodes".gaugeRnR."step".transition1[190] := ("Unit1.Em5.ControlNodes".gaugeRnR.sequence.status.currentStep = #JOB_1_STEP_90) AND "Unit1.Em5.ControlNodes".gaugeRnR.sequence.status.seqActive;
   IF ("Unit1.Em5.ControlNodes".gaugeRnR.sequence.status.currentStep = #JOB_1_STEP_90) AND "Unit1.Em5.ControlNodes".gaugeRnR.sequence.status.seqActive AND "Unit1.Em5.ControlNodes".gaugeRnR."step".transition1[190] THEN
       "Unit1.Em5.ControlNodes".gaugeRnR.sequence.status.nextStep := #STEP_IDLE;
   END_IF;
END_REGION

REGION Network 13: *************** JOB[2] Common Get Master Piece ************************
END_REGION

REGION Network 14: Step[201] : JOB[2] Condition
   RUNG wire#powerrail
      { S7_Templates := "SrcType := DInt" } EQ_Contact(in1 := "Unit1.Em5.ControlNodes".gaugeRnR.sequence.status.currentStep, in2 := #JOB_2_STEP_01)
      Contact( "Unit1.Em5.ControlNodes".gaugeRnR.sequence.status.seqActive )
      wire#w1
      Coil( "Unit1.Em5.ControlNodes".gaugeRnR."step".action1[201] )
   END_RUNG
   RUNG wire#w1
      Coil( "Unit1.Em5.ControlNodes".gaugeRnR."step".transition1[201] )
   END_RUNG
   RUNG wire#w1
      Contact( "Unit1.Em5.ControlNodes".gaugeRnR."step".transition1[201] )
      Move(in := #JOB_2_STEP_10, out1 => "Unit1.Em5.ControlNodes".gaugeRnR.sequence.status.nextStep)
   END_RUNG
   // the same network as SCL:
   "Unit1.Em5.ControlNodes".gaugeRnR."step".action1[201] := ("Unit1.Em5.ControlNodes".gaugeRnR.sequence.status.currentStep = #JOB_2_STEP_01) AND "Unit1.Em5.ControlNodes".gaugeRnR.sequence.status.seqActive;
   "Unit1.Em5.ControlNodes".gaugeRnR."step".transition1[201] := ("Unit1.Em5.ControlNodes".gaugeRnR.sequence.status.currentStep = #JOB_2_STEP_01) AND "Unit1.Em5.ControlNodes".gaugeRnR.sequence.status.seqActive;
   IF ("Unit1.Em5.ControlNodes".gaugeRnR.sequence.status.currentStep = #JOB_2_STEP_01) AND "Unit1.Em5.ControlNodes".gaugeRnR.sequence.status.seqActive AND "Unit1.Em5.ControlNodes".gaugeRnR."step".transition1[201] THEN
       "Unit1.Em5.ControlNodes".gaugeRnR.sequence.status.nextStep := #JOB_2_STEP_10;
   END_IF;
END_REGION

REGION Network 15: Step[210] : MainPnP1 Z-Axis Conveyor Down
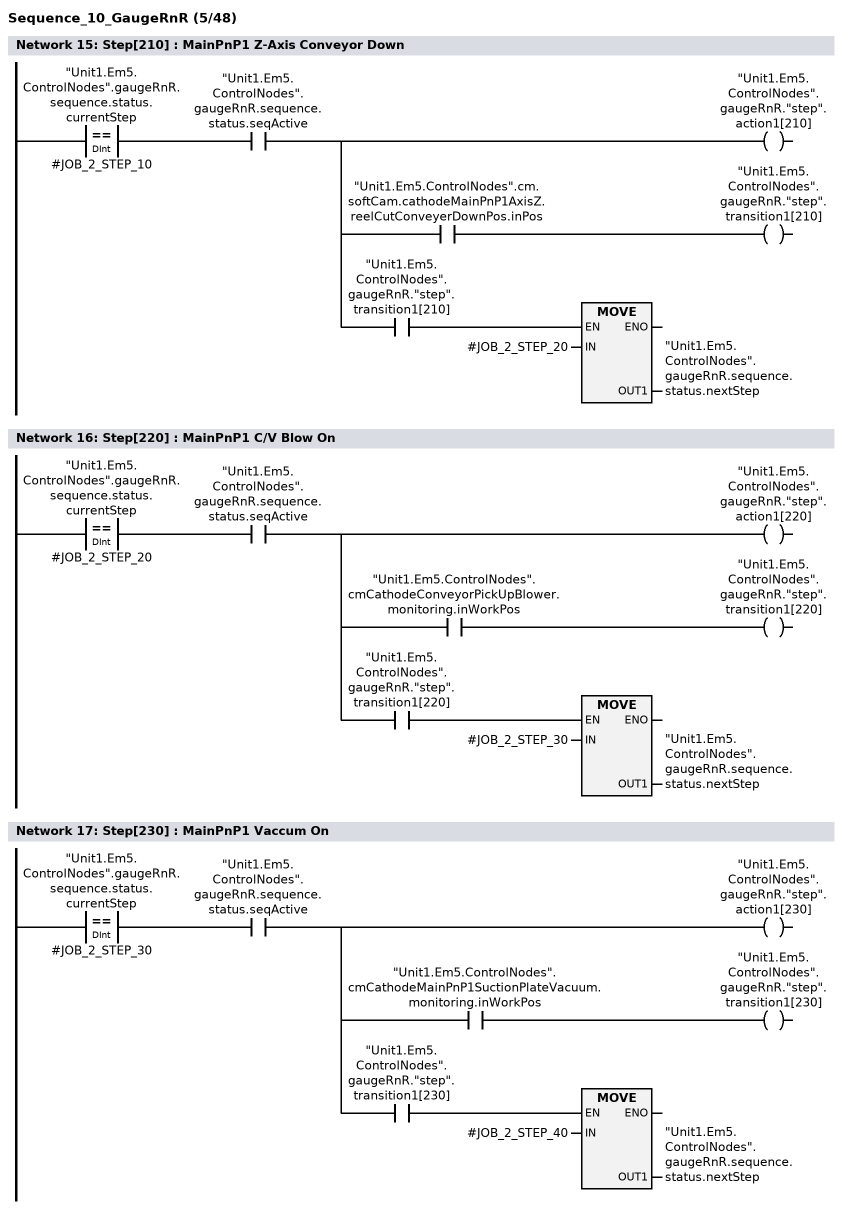
   RUNG wire#powerrail
      { S7_Templates := "SrcType := DInt" } EQ_Contact(in1 := "Unit1.Em5.ControlNodes".gaugeRnR.sequence.status.currentStep, in2 := #JOB_2_STEP_10)
      Contact( "Unit1.Em5.ControlNodes".gaugeRnR.sequence.status.seqActive )
      wire#w1
      Coil( "Unit1.Em5.ControlNodes".gaugeRnR."step".action1[210] )
   END_RUNG
   RUNG wire#w1
      Contact( "Unit1.Em5.ControlNodes".cm.softCam.cathodeMainPnP1AxisZ.reelCutConveyerDownPos.inPos )
      Coil( "Unit1.Em5.ControlNodes".gaugeRnR."step".transition1[210] )
   END_RUNG
   RUNG wire#w1
      Contact( "Unit1.Em5.ControlNodes".gaugeRnR."step".transition1[210] )
      Move(in := #JOB_2_STEP_20, out1 => "Unit1.Em5.ControlNodes".gaugeRnR.sequence.status.nextStep)
   END_RUNG
   // the same network as SCL:
   "Unit1.Em5.ControlNodes".gaugeRnR."step".action1[210] := ("Unit1.Em5.ControlNodes".gaugeRnR.sequence.status.currentStep = #JOB_2_STEP_10) AND "Unit1.Em5.ControlNodes".gaugeRnR.sequence.status.seqActive;
   "Unit1.Em5.ControlNodes".gaugeRnR."step".transition1[210] := ("Unit1.Em5.ControlNodes".gaugeRnR.sequence.status.currentStep = #JOB_2_STEP_10) AND "Unit1.Em5.ControlNodes".gaugeRnR.sequence.status.seqActive AND "Unit1.Em5.ControlNodes".cm.softCam.cathodeMainPnP1AxisZ.reelCutConveyerDownPos.inPos;
   IF ("Unit1.Em5.ControlNodes".gaugeRnR.sequence.status.currentStep = #JOB_2_STEP_10) AND "Unit1.Em5.ControlNodes".gaugeRnR.sequence.status.seqActive AND "Unit1.Em5.ControlNodes".gaugeRnR."step".transition1[210] THEN
       "Unit1.Em5.ControlNodes".gaugeRnR.sequence.status.nextStep := #JOB_2_STEP_20;
   END_IF;
END_REGION

REGION Network 16: Step[220] : MainPnP1 C/V Blow On
   RUNG wire#powerrail
      { S7_Templates := "SrcType := DInt" } EQ_Contact(in1 := "Unit1.Em5.ControlNodes".gaugeRnR.sequence.status.currentStep, in2 := #JOB_2_STEP_20)
      Contact( "Unit1.Em5.ControlNodes".gaugeRnR.sequence.status.seqActive )
      wire#w1
      Coil( "Unit1.Em5.ControlNodes".gaugeRnR."step".action1[220] )
   END_RUNG
   RUNG wire#w1
      Contact( "Unit1.Em5.ControlNodes".cmCathodeConveyorPickUpBlower.monitoring.inWorkPos )
      Coil( "Unit1.Em5.ControlNodes".gaugeRnR."step".transition1[220] )
   END_RUNG
   RUNG wire#w1
      Contact( "Unit1.Em5.ControlNodes".gaugeRnR."step".transition1[220] )
      Move(in := #JOB_2_STEP_30, out1 => "Unit1.Em5.ControlNodes".gaugeRnR.sequence.status.nextStep)
   END_RUNG
   // the same network as SCL:
   "Unit1.Em5.ControlNodes".gaugeRnR."step".action1[220] := ("Unit1.Em5.ControlNodes".gaugeRnR.sequence.status.currentStep = #JOB_2_STEP_20) AND "Unit1.Em5.ControlNodes".gaugeRnR.sequence.status.seqActive;
   "Unit1.Em5.ControlNodes".gaugeRnR."step".transition1[220] := ("Unit1.Em5.ControlNodes".gaugeRnR.sequence.status.currentStep = #JOB_2_STEP_20) AND "Unit1.Em5.ControlNodes".gaugeRnR.sequence.status.seqActive AND "Unit1.Em5.ControlNodes".cmCathodeConveyorPickUpBlower.monitoring.inWorkPos;
   IF ("Unit1.Em5.ControlNodes".gaugeRnR.sequence.status.currentStep = #JOB_2_STEP_20) AND "Unit1.Em5.ControlNodes".gaugeRnR.sequence.status.seqActive AND "Unit1.Em5.ControlNodes".gaugeRnR."step".transition1[220] THEN
       "Unit1.Em5.ControlNodes".gaugeRnR.sequence.status.nextStep := #JOB_2_STEP_30;
   END_IF;
END_REGION

REGION Network 17: Step[230] : MainPnP1 Vaccum On
   RUNG wire#powerrail
      { S7_Templates := "SrcType := DInt" } EQ_Contact(in1 := "Unit1.Em5.ControlNodes".gaugeRnR.sequence.status.currentStep, in2 := #JOB_2_STEP_30)
      Contact( "Unit1.Em5.ControlNodes".gaugeRnR.sequence.status.seqActive )
      wire#w1
      Coil( "Unit1.Em5.ControlNodes".gaugeRnR."step".action1[230] )
   END_RUNG
   RUNG wire#w1
      Contact( "Unit1.Em5.ControlNodes".cmCathodeMainPnP1SuctionPlateVacuum.monitoring.inWorkPos )
      Coil( "Unit1.Em5.ControlNodes".gaugeRnR."step".transition1[230] )
   END_RUNG
   RUNG wire#w1
      Contact( "Unit1.Em5.ControlNodes".gaugeRnR."step".transition1[230] )
      Move(in := #JOB_2_STEP_40, out1 => "Unit1.Em5.ControlNodes".gaugeRnR.sequence.status.nextStep)
   END_RUNG
   // the same network as SCL:
   "Unit1.Em5.ControlNodes".gaugeRnR."step".action1[230] := ("Unit1.Em5.ControlNodes".gaugeRnR.sequence.status.currentStep = #JOB_2_STEP_30) AND "Unit1.Em5.ControlNodes".gaugeRnR.sequence.status.seqActive;
   "Unit1.Em5.ControlNodes".gaugeRnR."step".transition1[230] := ("Unit1.Em5.ControlNodes".gaugeRnR.sequence.status.currentStep = #JOB_2_STEP_30) AND "Unit1.Em5.ControlNodes".gaugeRnR.sequence.status.seqActive AND "Unit1.Em5.ControlNodes".cmCathodeMainPnP1SuctionPlateVacuum.monitoring.inWorkPos;
   IF ("Unit1.Em5.ControlNodes".gaugeRnR.sequence.status.currentStep = #JOB_2_STEP_30) AND "Unit1.Em5.ControlNodes".gaugeRnR.sequence.status.seqActive AND "Unit1.Em5.ControlNodes".gaugeRnR."step".transition1[230] THEN
       "Unit1.Em5.ControlNodes".gaugeRnR.sequence.status.nextStep := #JOB_2_STEP_40;
   END_IF;
END_REGION

REGION Network 18: Step[240] : MainPnP1 C/V Blow Off
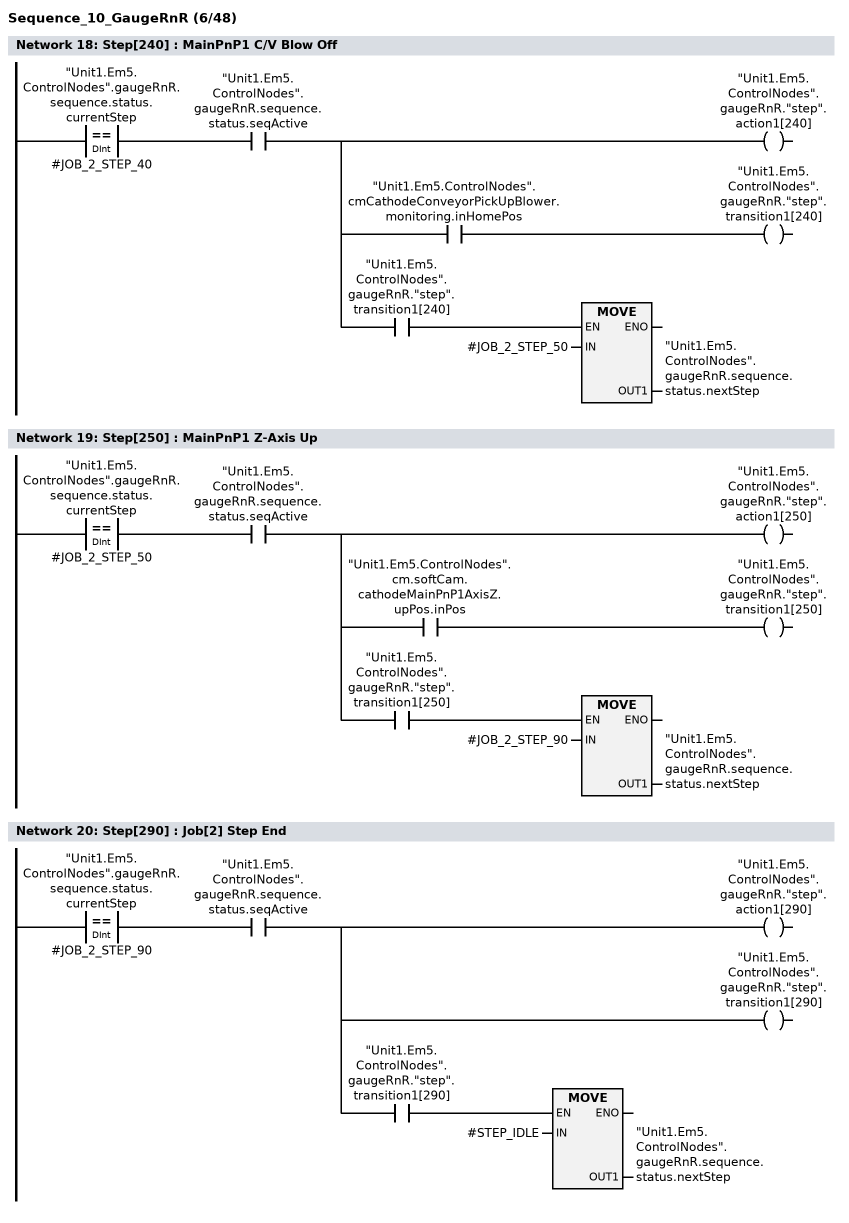
   RUNG wire#powerrail
      { S7_Templates := "SrcType := DInt" } EQ_Contact(in1 := "Unit1.Em5.ControlNodes".gaugeRnR.sequence.status.currentStep, in2 := #JOB_2_STEP_40)
      Contact( "Unit1.Em5.ControlNodes".gaugeRnR.sequence.status.seqActive )
      wire#w1
      Coil( "Unit1.Em5.ControlNodes".gaugeRnR."step".action1[240] )
   END_RUNG
   RUNG wire#w1
      Contact( "Unit1.Em5.ControlNodes".cmCathodeConveyorPickUpBlower.monitoring.inHomePos )
      Coil( "Unit1.Em5.ControlNodes".gaugeRnR."step".transition1[240] )
   END_RUNG
   RUNG wire#w1
      Contact( "Unit1.Em5.ControlNodes".gaugeRnR."step".transition1[240] )
      Move(in := #JOB_2_STEP_50, out1 => "Unit1.Em5.ControlNodes".gaugeRnR.sequence.status.nextStep)
   END_RUNG
   // the same network as SCL:
   "Unit1.Em5.ControlNodes".gaugeRnR."step".action1[240] := ("Unit1.Em5.ControlNodes".gaugeRnR.sequence.status.currentStep = #JOB_2_STEP_40) AND "Unit1.Em5.ControlNodes".gaugeRnR.sequence.status.seqActive;
   "Unit1.Em5.ControlNodes".gaugeRnR."step".transition1[240] := ("Unit1.Em5.ControlNodes".gaugeRnR.sequence.status.currentStep = #JOB_2_STEP_40) AND "Unit1.Em5.ControlNodes".gaugeRnR.sequence.status.seqActive AND "Unit1.Em5.ControlNodes".cmCathodeConveyorPickUpBlower.monitoring.inHomePos;
   IF ("Unit1.Em5.ControlNodes".gaugeRnR.sequence.status.currentStep = #JOB_2_STEP_40) AND "Unit1.Em5.ControlNodes".gaugeRnR.sequence.status.seqActive AND "Unit1.Em5.ControlNodes".gaugeRnR."step".transition1[240] THEN
       "Unit1.Em5.ControlNodes".gaugeRnR.sequence.status.nextStep := #JOB_2_STEP_50;
   END_IF;
END_REGION

REGION Network 19: Step[250] : MainPnP1 Z-Axis Up
   RUNG wire#powerrail
      { S7_Templates := "SrcType := DInt" } EQ_Contact(in1 := "Unit1.Em5.ControlNodes".gaugeRnR.sequence.status.currentStep, in2 := #JOB_2_STEP_50)
      Contact( "Unit1.Em5.ControlNodes".gaugeRnR.sequence.status.seqActive )
      wire#w1
      Coil( "Unit1.Em5.ControlNodes".gaugeRnR."step".action1[250] )
   END_RUNG
   RUNG wire#w1
      Contact( "Unit1.Em5.ControlNodes".cm.softCam.cathodeMainPnP1AxisZ.upPos.inPos )
      Coil( "Unit1.Em5.ControlNodes".gaugeRnR."step".transition1[250] )
   END_RUNG
   RUNG wire#w1
      Contact( "Unit1.Em5.ControlNodes".gaugeRnR."step".transition1[250] )
      Move(in := #JOB_2_STEP_90, out1 => "Unit1.Em5.ControlNodes".gaugeRnR.sequence.status.nextStep)
   END_RUNG
   // the same network as SCL:
   "Unit1.Em5.ControlNodes".gaugeRnR."step".action1[250] := ("Unit1.Em5.ControlNodes".gaugeRnR.sequence.status.currentStep = #JOB_2_STEP_50) AND "Unit1.Em5.ControlNodes".gaugeRnR.sequence.status.seqActive;
   "Unit1.Em5.ControlNodes".gaugeRnR."step".transition1[250] := ("Unit1.Em5.ControlNodes".gaugeRnR.sequence.status.currentStep = #JOB_2_STEP_50) AND "Unit1.Em5.ControlNodes".gaugeRnR.sequence.status.seqActive AND "Unit1.Em5.ControlNodes".cm.softCam.cathodeMainPnP1AxisZ.upPos.inPos;
   IF ("Unit1.Em5.ControlNodes".gaugeRnR.sequence.status.currentStep = #JOB_2_STEP_50) AND "Unit1.Em5.ControlNodes".gaugeRnR.sequence.status.seqActive AND "Unit1.Em5.ControlNodes".gaugeRnR."step".transition1[250] THEN
       "Unit1.Em5.ControlNodes".gaugeRnR.sequence.status.nextStep := #JOB_2_STEP_90;
   END_IF;
END_REGION

REGION Network 20: Step[290] : Job[2] Step End
   RUNG wire#powerrail
      { S7_Templates := "SrcType := DInt" } EQ_Contact(in1 := "Unit1.Em5.ControlNodes".gaugeRnR.sequence.status.currentStep, in2 := #JOB_2_STEP_90)
      Contact( "Unit1.Em5.ControlNodes".gaugeRnR.sequence.status.seqActive )
      wire#w1
      Coil( "Unit1.Em5.ControlNodes".gaugeRnR."step".action1[290] )
   END_RUNG
   RUNG wire#w1
      Coil( "Unit1.Em5.ControlNodes".gaugeRnR."step".transition1[290] )
   END_RUNG
   RUNG wire#w1
      Contact( "Unit1.Em5.ControlNodes".gaugeRnR."step".transition1[290] )
      Move(in := #STEP_IDLE, out1 => "Unit1.Em5.ControlNodes".gaugeRnR.sequence.status.nextStep)
   END_RUNG
   // the same network as SCL:
   "Unit1.Em5.ControlNodes".gaugeRnR."step".action1[290] := ("Unit1.Em5.ControlNodes".gaugeRnR.sequence.status.currentStep = #JOB_2_STEP_90) AND "Unit1.Em5.ControlNodes".gaugeRnR.sequence.status.seqActive;
   "Unit1.Em5.ControlNodes".gaugeRnR."step".transition1[290] := ("Unit1.Em5.ControlNodes".gaugeRnR.sequence.status.currentStep = #JOB_2_STEP_90) AND "Unit1.Em5.ControlNodes".gaugeRnR.sequence.status.seqActive;
   IF ("Unit1.Em5.ControlNodes".gaugeRnR.sequence.status.currentStep = #JOB_2_STEP_90) AND "Unit1.Em5.ControlNodes".gaugeRnR.sequence.status.seqActive AND "Unit1.Em5.ControlNodes".gaugeRnR."step".transition1[290] THEN
       "Unit1.Em5.ControlNodes".gaugeRnR.sequence.status.nextStep := #STEP_IDLE;
   END_IF;
END_REGION

REGION Network 21: *************** JOB[3] Common MainPnP Move AlignTable / StackTable ************************
END_REGION

REGION Network 22: Step[301] : JOB[3] Condition
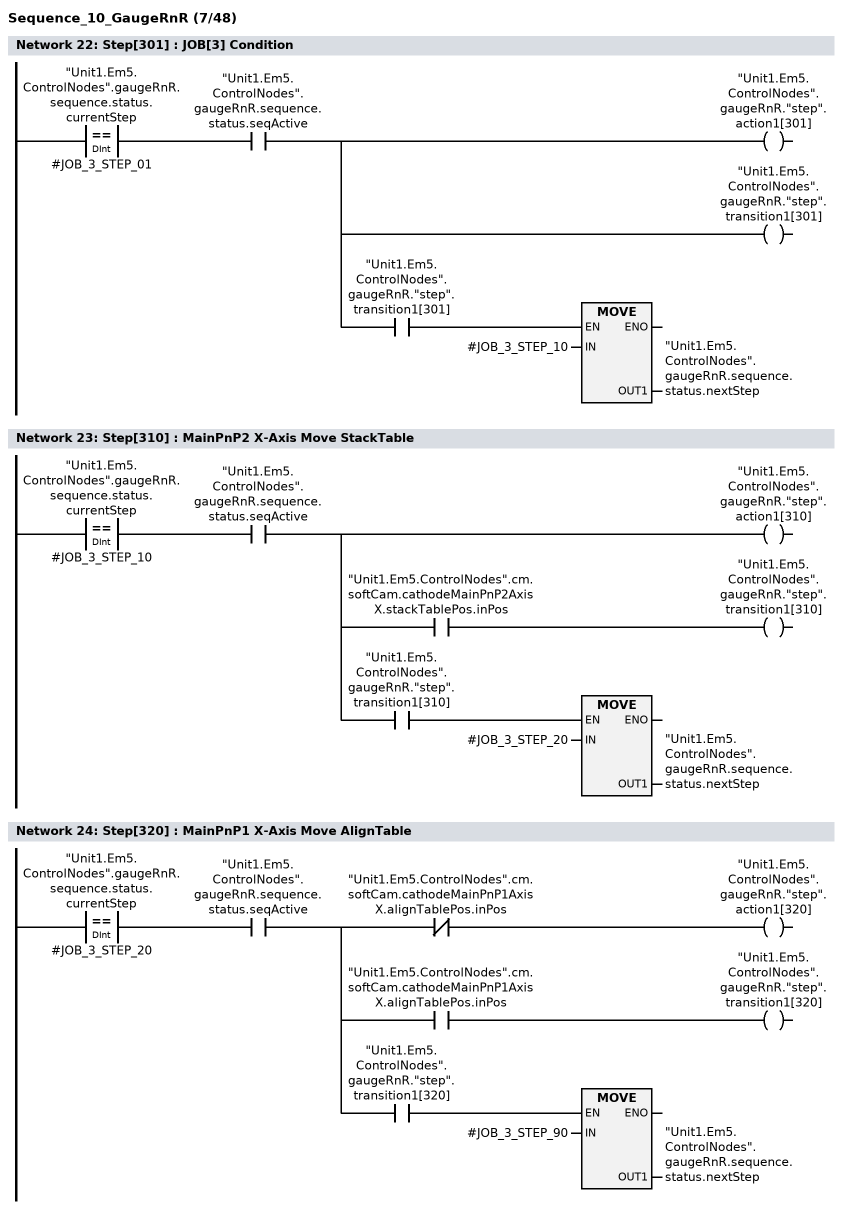
   RUNG wire#powerrail
      { S7_Templates := "SrcType := DInt" } EQ_Contact(in1 := "Unit1.Em5.ControlNodes".gaugeRnR.sequence.status.currentStep, in2 := #JOB_3_STEP_01)
      Contact( "Unit1.Em5.ControlNodes".gaugeRnR.sequence.status.seqActive )
      wire#w1
      Coil( "Unit1.Em5.ControlNodes".gaugeRnR."step".action1[301] )
   END_RUNG
   RUNG wire#w1
      Coil( "Unit1.Em5.ControlNodes".gaugeRnR."step".transition1[301] )
   END_RUNG
   RUNG wire#w1
      Contact( "Unit1.Em5.ControlNodes".gaugeRnR."step".transition1[301] )
      Move(in := #JOB_3_STEP_10, out1 => "Unit1.Em5.ControlNodes".gaugeRnR.sequence.status.nextStep)
   END_RUNG
   // the same network as SCL:
   "Unit1.Em5.ControlNodes".gaugeRnR."step".action1[301] := ("Unit1.Em5.ControlNodes".gaugeRnR.sequence.status.currentStep = #JOB_3_STEP_01) AND "Unit1.Em5.ControlNodes".gaugeRnR.sequence.status.seqActive;
   "Unit1.Em5.ControlNodes".gaugeRnR."step".transition1[301] := ("Unit1.Em5.ControlNodes".gaugeRnR.sequence.status.currentStep = #JOB_3_STEP_01) AND "Unit1.Em5.ControlNodes".gaugeRnR.sequence.status.seqActive;
   IF ("Unit1.Em5.ControlNodes".gaugeRnR.sequence.status.currentStep = #JOB_3_STEP_01) AND "Unit1.Em5.ControlNodes".gaugeRnR.sequence.status.seqActive AND "Unit1.Em5.ControlNodes".gaugeRnR."step".transition1[301] THEN
       "Unit1.Em5.ControlNodes".gaugeRnR.sequence.status.nextStep := #JOB_3_STEP_10;
   END_IF;
END_REGION

REGION Network 23: Step[310] : MainPnP2 X-Axis Move StackTable
   RUNG wire#powerrail
      { S7_Templates := "SrcType := DInt" } EQ_Contact(in1 := "Unit1.Em5.ControlNodes".gaugeRnR.sequence.status.currentStep, in2 := #JOB_3_STEP_10)
      Contact( "Unit1.Em5.ControlNodes".gaugeRnR.sequence.status.seqActive )
      wire#w1
      Coil( "Unit1.Em5.ControlNodes".gaugeRnR."step".action1[310] )
   END_RUNG
   RUNG wire#w1
      Contact( "Unit1.Em5.ControlNodes".cm.softCam.cathodeMainPnP2AxisX.stackTablePos.inPos )
      Coil( "Unit1.Em5.ControlNodes".gaugeRnR."step".transition1[310] )
   END_RUNG
   RUNG wire#w1
      Contact( "Unit1.Em5.ControlNodes".gaugeRnR."step".transition1[310] )
      Move(in := #JOB_3_STEP_20, out1 => "Unit1.Em5.ControlNodes".gaugeRnR.sequence.status.nextStep)
   END_RUNG
   // the same network as SCL:
   "Unit1.Em5.ControlNodes".gaugeRnR."step".action1[310] := ("Unit1.Em5.ControlNodes".gaugeRnR.sequence.status.currentStep = #JOB_3_STEP_10) AND "Unit1.Em5.ControlNodes".gaugeRnR.sequence.status.seqActive;
   "Unit1.Em5.ControlNodes".gaugeRnR."step".transition1[310] := ("Unit1.Em5.ControlNodes".gaugeRnR.sequence.status.currentStep = #JOB_3_STEP_10) AND "Unit1.Em5.ControlNodes".gaugeRnR.sequence.status.seqActive AND "Unit1.Em5.ControlNodes".cm.softCam.cathodeMainPnP2AxisX.stackTablePos.inPos;
   IF ("Unit1.Em5.ControlNodes".gaugeRnR.sequence.status.currentStep = #JOB_3_STEP_10) AND "Unit1.Em5.ControlNodes".gaugeRnR.sequence.status.seqActive AND "Unit1.Em5.ControlNodes".gaugeRnR."step".transition1[310] THEN
       "Unit1.Em5.ControlNodes".gaugeRnR.sequence.status.nextStep := #JOB_3_STEP_20;
   END_IF;
END_REGION

REGION Network 24: Step[320] : MainPnP1 X-Axis Move AlignTable
   RUNG wire#powerrail
      { S7_Templates := "SrcType := DInt" } EQ_Contact(in1 := "Unit1.Em5.ControlNodes".gaugeRnR.sequence.status.currentStep, in2 := #JOB_3_STEP_20)
      Contact( "Unit1.Em5.ControlNodes".gaugeRnR.sequence.status.seqActive )
      wire#w1
      I_Contact( "Unit1.Em5.ControlNodes".cm.softCam.cathodeMainPnP1AxisX.alignTablePos.inPos )
      Coil( "Unit1.Em5.ControlNodes".gaugeRnR."step".action1[320] )
   END_RUNG
   RUNG wire#w1
      Contact( "Unit1.Em5.ControlNodes".cm.softCam.cathodeMainPnP1AxisX.alignTablePos.inPos )
      Coil( "Unit1.Em5.ControlNodes".gaugeRnR."step".transition1[320] )
   END_RUNG
   RUNG wire#w1
      Contact( "Unit1.Em5.ControlNodes".gaugeRnR."step".transition1[320] )
      Move(in := #JOB_3_STEP_90, out1 => "Unit1.Em5.ControlNodes".gaugeRnR.sequence.status.nextStep)
   END_RUNG
   // the same network as SCL:
   #_w1 := ("Unit1.Em5.ControlNodes".gaugeRnR.sequence.status.currentStep = #JOB_3_STEP_20) AND "Unit1.Em5.ControlNodes".gaugeRnR.sequence.status.seqActive;
   "Unit1.Em5.ControlNodes".gaugeRnR."step".action1[320] := #_w1 AND NOT "Unit1.Em5.ControlNodes".cm.softCam.cathodeMainPnP1AxisX.alignTablePos.inPos;
   "Unit1.Em5.ControlNodes".gaugeRnR."step".transition1[320] := #_w1 AND "Unit1.Em5.ControlNodes".cm.softCam.cathodeMainPnP1AxisX.alignTablePos.inPos;
   IF #_w1 AND "Unit1.Em5.ControlNodes".gaugeRnR."step".transition1[320] THEN
       "Unit1.Em5.ControlNodes".gaugeRnR.sequence.status.nextStep := #JOB_3_STEP_90;
   END_IF;
END_REGION

REGION Network 25: Step[390] : Job[3] Step End
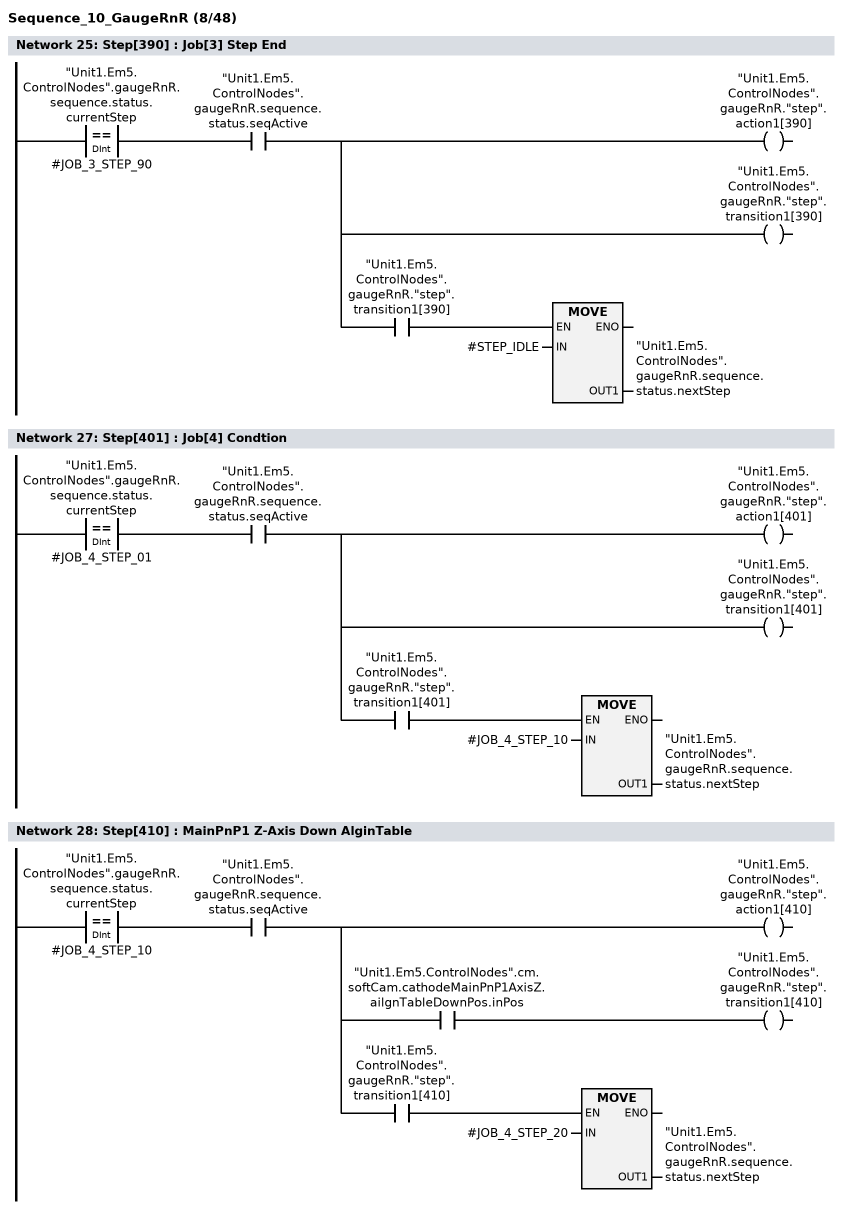
   RUNG wire#powerrail
      { S7_Templates := "SrcType := DInt" } EQ_Contact(in1 := "Unit1.Em5.ControlNodes".gaugeRnR.sequence.status.currentStep, in2 := #JOB_3_STEP_90)
      Contact( "Unit1.Em5.ControlNodes".gaugeRnR.sequence.status.seqActive )
      wire#w1
      Coil( "Unit1.Em5.ControlNodes".gaugeRnR."step".action1[390] )
   END_RUNG
   RUNG wire#w1
      Coil( "Unit1.Em5.ControlNodes".gaugeRnR."step".transition1[390] )
   END_RUNG
   RUNG wire#w1
      Contact( "Unit1.Em5.ControlNodes".gaugeRnR."step".transition1[390] )
      Move(in := #STEP_IDLE, out1 => "Unit1.Em5.ControlNodes".gaugeRnR.sequence.status.nextStep)
   END_RUNG
   // the same network as SCL:
   "Unit1.Em5.ControlNodes".gaugeRnR."step".action1[390] := ("Unit1.Em5.ControlNodes".gaugeRnR.sequence.status.currentStep = #JOB_3_STEP_90) AND "Unit1.Em5.ControlNodes".gaugeRnR.sequence.status.seqActive;
   "Unit1.Em5.ControlNodes".gaugeRnR."step".transition1[390] := ("Unit1.Em5.ControlNodes".gaugeRnR.sequence.status.currentStep = #JOB_3_STEP_90) AND "Unit1.Em5.ControlNodes".gaugeRnR.sequence.status.seqActive;
   IF ("Unit1.Em5.ControlNodes".gaugeRnR.sequence.status.currentStep = #JOB_3_STEP_90) AND "Unit1.Em5.ControlNodes".gaugeRnR.sequence.status.seqActive AND "Unit1.Em5.ControlNodes".gaugeRnR."step".transition1[390] THEN
       "Unit1.Em5.ControlNodes".gaugeRnR.sequence.status.nextStep := #STEP_IDLE;
   END_IF;
END_REGION

REGION Network 26: *************** JOB[4] Common MainPnP1 To AlignTable************************
END_REGION

REGION Network 27: Step[401] : Job[4] Condtion
   RUNG wire#powerrail
      { S7_Templates := "SrcType := DInt" } EQ_Contact(in1 := "Unit1.Em5.ControlNodes".gaugeRnR.sequence.status.currentStep, in2 := #JOB_4_STEP_01)
      Contact( "Unit1.Em5.ControlNodes".gaugeRnR.sequence.status.seqActive )
      wire#w1
      Coil( "Unit1.Em5.ControlNodes".gaugeRnR."step".action1[401] )
   END_RUNG
   RUNG wire#w1
      Coil( "Unit1.Em5.ControlNodes".gaugeRnR."step".transition1[401] )
   END_RUNG
   RUNG wire#w1
      Contact( "Unit1.Em5.ControlNodes".gaugeRnR."step".transition1[401] )
      Move(in := #JOB_4_STEP_10, out1 => "Unit1.Em5.ControlNodes".gaugeRnR.sequence.status.nextStep)
   END_RUNG
   // the same network as SCL:
   "Unit1.Em5.ControlNodes".gaugeRnR."step".action1[401] := ("Unit1.Em5.ControlNodes".gaugeRnR.sequence.status.currentStep = #JOB_4_STEP_01) AND "Unit1.Em5.ControlNodes".gaugeRnR.sequence.status.seqActive;
   "Unit1.Em5.ControlNodes".gaugeRnR."step".transition1[401] := ("Unit1.Em5.ControlNodes".gaugeRnR.sequence.status.currentStep = #JOB_4_STEP_01) AND "Unit1.Em5.ControlNodes".gaugeRnR.sequence.status.seqActive;
   IF ("Unit1.Em5.ControlNodes".gaugeRnR.sequence.status.currentStep = #JOB_4_STEP_01) AND "Unit1.Em5.ControlNodes".gaugeRnR.sequence.status.seqActive AND "Unit1.Em5.ControlNodes".gaugeRnR."step".transition1[401] THEN
       "Unit1.Em5.ControlNodes".gaugeRnR.sequence.status.nextStep := #JOB_4_STEP_10;
   END_IF;
END_REGION

REGION Network 28: Step[410] : MainPnP1 Z-Axis Down AlginTable
   RUNG wire#powerrail
      { S7_Templates := "SrcType := DInt" } EQ_Contact(in1 := "Unit1.Em5.ControlNodes".gaugeRnR.sequence.status.currentStep, in2 := #JOB_4_STEP_10)
      Contact( "Unit1.Em5.ControlNodes".gaugeRnR.sequence.status.seqActive )
      wire#w1
      Coil( "Unit1.Em5.ControlNodes".gaugeRnR."step".action1[410] )
   END_RUNG
   RUNG wire#w1
      Contact( "Unit1.Em5.ControlNodes".cm.softCam.cathodeMainPnP1AxisZ.ailgnTableDownPos.inPos )
      Coil( "Unit1.Em5.ControlNodes".gaugeRnR."step".transition1[410] )
   END_RUNG
   RUNG wire#w1
      Contact( "Unit1.Em5.ControlNodes".gaugeRnR."step".transition1[410] )
      Move(in := #JOB_4_STEP_20, out1 => "Unit1.Em5.ControlNodes".gaugeRnR.sequence.status.nextStep)
   END_RUNG
   // the same network as SCL:
   "Unit1.Em5.ControlNodes".gaugeRnR."step".action1[410] := ("Unit1.Em5.ControlNodes".gaugeRnR.sequence.status.currentStep = #JOB_4_STEP_10) AND "Unit1.Em5.ControlNodes".gaugeRnR.sequence.status.seqActive;
   "Unit1.Em5.ControlNodes".gaugeRnR."step".transition1[410] := ("Unit1.Em5.ControlNodes".gaugeRnR.sequence.status.currentStep = #JOB_4_STEP_10) AND "Unit1.Em5.ControlNodes".gaugeRnR.sequence.status.seqActive AND "Unit1.Em5.ControlNodes".cm.softCam.cathodeMainPnP1AxisZ.ailgnTableDownPos.inPos;
   IF ("Unit1.Em5.ControlNodes".gaugeRnR.sequence.status.currentStep = #JOB_4_STEP_10) AND "Unit1.Em5.ControlNodes".gaugeRnR.sequence.status.seqActive AND "Unit1.Em5.ControlNodes".gaugeRnR."step".transition1[410] THEN
       "Unit1.Em5.ControlNodes".gaugeRnR.sequence.status.nextStep := #JOB_4_STEP_20;
   END_IF;
END_REGION

REGION Network 29: Step[420] : MainPnP1 1 Vaccum Off
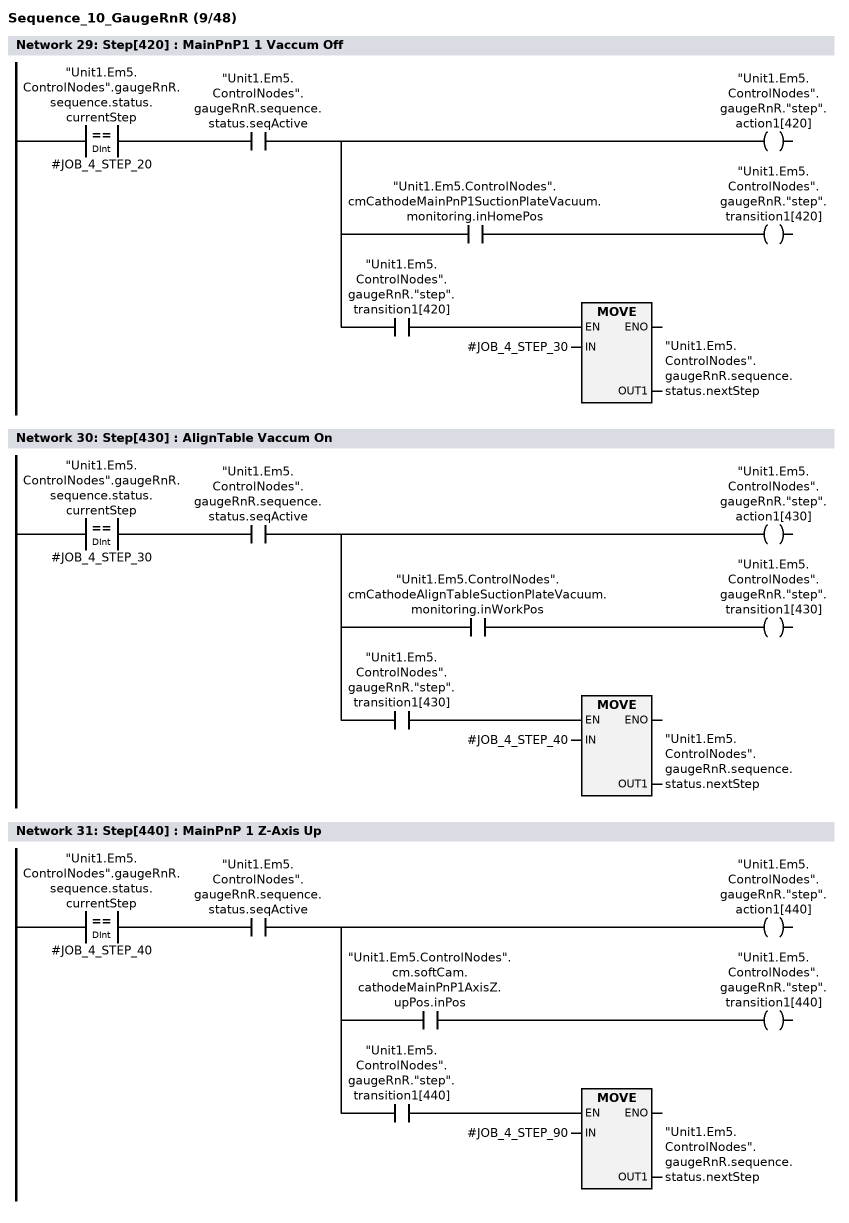
   RUNG wire#powerrail
      { S7_Templates := "SrcType := DInt" } EQ_Contact(in1 := "Unit1.Em5.ControlNodes".gaugeRnR.sequence.status.currentStep, in2 := #JOB_4_STEP_20)
      Contact( "Unit1.Em5.ControlNodes".gaugeRnR.sequence.status.seqActive )
      wire#w1
      Coil( "Unit1.Em5.ControlNodes".gaugeRnR."step".action1[420] )
   END_RUNG
   RUNG wire#w1
      Contact( "Unit1.Em5.ControlNodes".cmCathodeMainPnP1SuctionPlateVacuum.monitoring.inHomePos )
      Coil( "Unit1.Em5.ControlNodes".gaugeRnR."step".transition1[420] )
   END_RUNG
   RUNG wire#w1
      Contact( "Unit1.Em5.ControlNodes".gaugeRnR."step".transition1[420] )
      Move(in := #JOB_4_STEP_30, out1 => "Unit1.Em5.ControlNodes".gaugeRnR.sequence.status.nextStep)
   END_RUNG
   // the same network as SCL:
   "Unit1.Em5.ControlNodes".gaugeRnR."step".action1[420] := ("Unit1.Em5.ControlNodes".gaugeRnR.sequence.status.currentStep = #JOB_4_STEP_20) AND "Unit1.Em5.ControlNodes".gaugeRnR.sequence.status.seqActive;
   "Unit1.Em5.ControlNodes".gaugeRnR."step".transition1[420] := ("Unit1.Em5.ControlNodes".gaugeRnR.sequence.status.currentStep = #JOB_4_STEP_20) AND "Unit1.Em5.ControlNodes".gaugeRnR.sequence.status.seqActive AND "Unit1.Em5.ControlNodes".cmCathodeMainPnP1SuctionPlateVacuum.monitoring.inHomePos;
   IF ("Unit1.Em5.ControlNodes".gaugeRnR.sequence.status.currentStep = #JOB_4_STEP_20) AND "Unit1.Em5.ControlNodes".gaugeRnR.sequence.status.seqActive AND "Unit1.Em5.ControlNodes".gaugeRnR."step".transition1[420] THEN
       "Unit1.Em5.ControlNodes".gaugeRnR.sequence.status.nextStep := #JOB_4_STEP_30;
   END_IF;
END_REGION

REGION Network 30: Step[430] : AlignTable Vaccum On
   RUNG wire#powerrail
      { S7_Templates := "SrcType := DInt" } EQ_Contact(in1 := "Unit1.Em5.ControlNodes".gaugeRnR.sequence.status.currentStep, in2 := #JOB_4_STEP_30)
      Contact( "Unit1.Em5.ControlNodes".gaugeRnR.sequence.status.seqActive )
      wire#w1
      Coil( "Unit1.Em5.ControlNodes".gaugeRnR."step".action1[430] )
   END_RUNG
   RUNG wire#w1
      Contact( "Unit1.Em5.ControlNodes".cmCathodeAlignTableSuctionPlateVacuum.monitoring.inWorkPos )
      Coil( "Unit1.Em5.ControlNodes".gaugeRnR."step".transition1[430] )
   END_RUNG
   RUNG wire#w1
      Contact( "Unit1.Em5.ControlNodes".gaugeRnR."step".transition1[430] )
      Move(in := #JOB_4_STEP_40, out1 => "Unit1.Em5.ControlNodes".gaugeRnR.sequence.status.nextStep)
   END_RUNG
   // the same network as SCL:
   "Unit1.Em5.ControlNodes".gaugeRnR."step".action1[430] := ("Unit1.Em5.ControlNodes".gaugeRnR.sequence.status.currentStep = #JOB_4_STEP_30) AND "Unit1.Em5.ControlNodes".gaugeRnR.sequence.status.seqActive;
   "Unit1.Em5.ControlNodes".gaugeRnR."step".transition1[430] := ("Unit1.Em5.ControlNodes".gaugeRnR.sequence.status.currentStep = #JOB_4_STEP_30) AND "Unit1.Em5.ControlNodes".gaugeRnR.sequence.status.seqActive AND "Unit1.Em5.ControlNodes".cmCathodeAlignTableSuctionPlateVacuum.monitoring.inWorkPos;
   IF ("Unit1.Em5.ControlNodes".gaugeRnR.sequence.status.currentStep = #JOB_4_STEP_30) AND "Unit1.Em5.ControlNodes".gaugeRnR.sequence.status.seqActive AND "Unit1.Em5.ControlNodes".gaugeRnR."step".transition1[430] THEN
       "Unit1.Em5.ControlNodes".gaugeRnR.sequence.status.nextStep := #JOB_4_STEP_40;
   END_IF;
END_REGION

REGION Network 31: Step[440] : MainPnP 1 Z-Axis Up
   RUNG wire#powerrail
      { S7_Templates := "SrcType := DInt" } EQ_Contact(in1 := "Unit1.Em5.ControlNodes".gaugeRnR.sequence.status.currentStep, in2 := #JOB_4_STEP_40)
      Contact( "Unit1.Em5.ControlNodes".gaugeRnR.sequence.status.seqActive )
      wire#w1
      Coil( "Unit1.Em5.ControlNodes".gaugeRnR."step".action1[440] )
   END_RUNG
   RUNG wire#w1
      Contact( "Unit1.Em5.ControlNodes".cm.softCam.cathodeMainPnP1AxisZ.upPos.inPos )
      Coil( "Unit1.Em5.ControlNodes".gaugeRnR."step".transition1[440] )
   END_RUNG
   RUNG wire#w1
      Contact( "Unit1.Em5.ControlNodes".gaugeRnR."step".transition1[440] )
      Move(in := #JOB_4_STEP_90, out1 => "Unit1.Em5.ControlNodes".gaugeRnR.sequence.status.nextStep)
   END_RUNG
   // the same network as SCL:
   "Unit1.Em5.ControlNodes".gaugeRnR."step".action1[440] := ("Unit1.Em5.ControlNodes".gaugeRnR.sequence.status.currentStep = #JOB_4_STEP_40) AND "Unit1.Em5.ControlNodes".gaugeRnR.sequence.status.seqActive;
   "Unit1.Em5.ControlNodes".gaugeRnR."step".transition1[440] := ("Unit1.Em5.ControlNodes".gaugeRnR.sequence.status.currentStep = #JOB_4_STEP_40) AND "Unit1.Em5.ControlNodes".gaugeRnR.sequence.status.seqActive AND "Unit1.Em5.ControlNodes".cm.softCam.cathodeMainPnP1AxisZ.upPos.inPos;
   IF ("Unit1.Em5.ControlNodes".gaugeRnR.sequence.status.currentStep = #JOB_4_STEP_40) AND "Unit1.Em5.ControlNodes".gaugeRnR.sequence.status.seqActive AND "Unit1.Em5.ControlNodes".gaugeRnR."step".transition1[440] THEN
       "Unit1.Em5.ControlNodes".gaugeRnR.sequence.status.nextStep := #JOB_4_STEP_90;
   END_IF;
END_REGION

REGION Network 32: Step[490] : Job[4] Step End
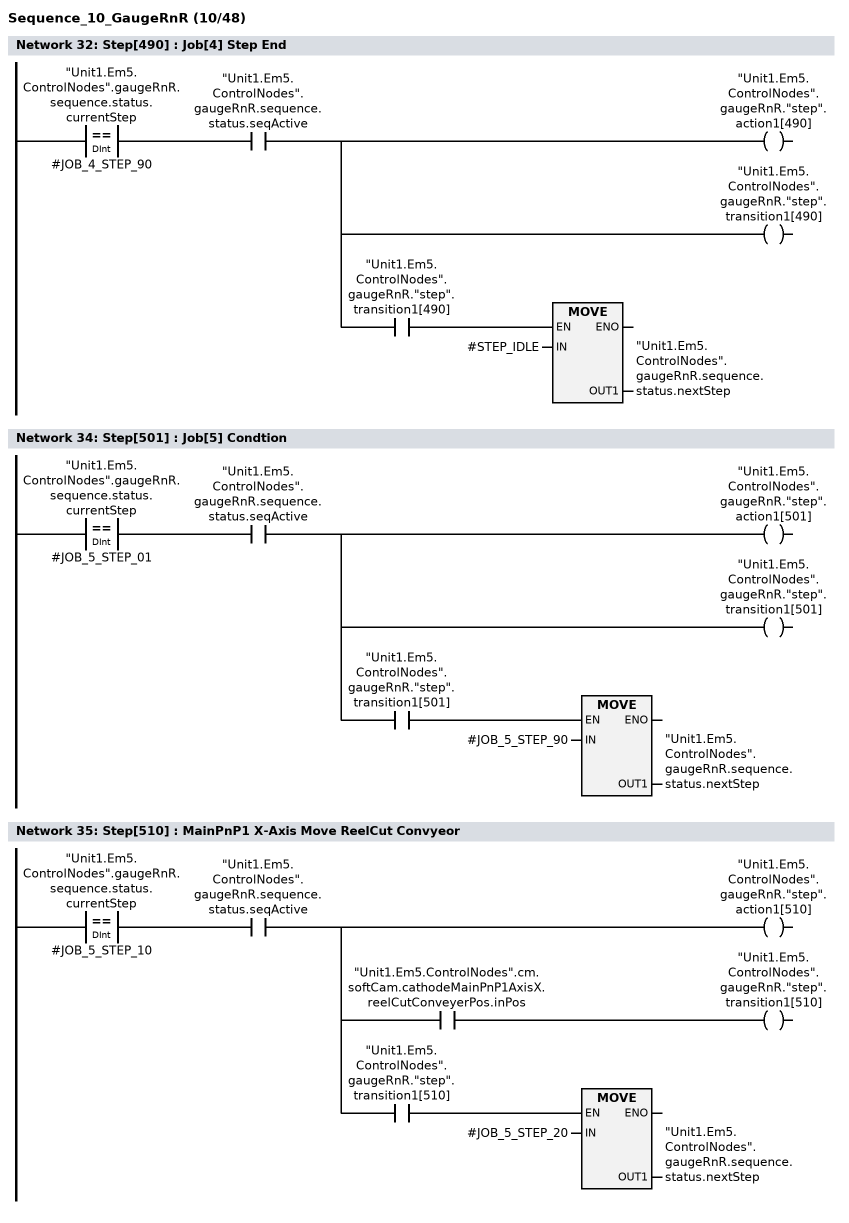
   RUNG wire#powerrail
      { S7_Templates := "SrcType := DInt" } EQ_Contact(in1 := "Unit1.Em5.ControlNodes".gaugeRnR.sequence.status.currentStep, in2 := #JOB_4_STEP_90)
      Contact( "Unit1.Em5.ControlNodes".gaugeRnR.sequence.status.seqActive )
      wire#w1
      Coil( "Unit1.Em5.ControlNodes".gaugeRnR."step".action1[490] )
   END_RUNG
   RUNG wire#w1
      Coil( "Unit1.Em5.ControlNodes".gaugeRnR."step".transition1[490] )
   END_RUNG
   RUNG wire#w1
      Contact( "Unit1.Em5.ControlNodes".gaugeRnR."step".transition1[490] )
      Move(in := #STEP_IDLE, out1 => "Unit1.Em5.ControlNodes".gaugeRnR.sequence.status.nextStep)
   END_RUNG
   // the same network as SCL:
   "Unit1.Em5.ControlNodes".gaugeRnR."step".action1[490] := ("Unit1.Em5.ControlNodes".gaugeRnR.sequence.status.currentStep = #JOB_4_STEP_90) AND "Unit1.Em5.ControlNodes".gaugeRnR.sequence.status.seqActive;
   "Unit1.Em5.ControlNodes".gaugeRnR."step".transition1[490] := ("Unit1.Em5.ControlNodes".gaugeRnR.sequence.status.currentStep = #JOB_4_STEP_90) AND "Unit1.Em5.ControlNodes".gaugeRnR.sequence.status.seqActive;
   IF ("Unit1.Em5.ControlNodes".gaugeRnR.sequence.status.currentStep = #JOB_4_STEP_90) AND "Unit1.Em5.ControlNodes".gaugeRnR.sequence.status.seqActive AND "Unit1.Em5.ControlNodes".gaugeRnR."step".transition1[490] THEN
       "Unit1.Em5.ControlNodes".gaugeRnR.sequence.status.nextStep := #STEP_IDLE;
   END_IF;
END_REGION

REGION Network 33: *************** JOB[5] Common MainPnP Move ReelCut Convyeor / AlignTable************************
END_REGION

REGION Network 34: Step[501] : Job[5] Condtion
   RUNG wire#powerrail
      { S7_Templates := "SrcType := DInt" } EQ_Contact(in1 := "Unit1.Em5.ControlNodes".gaugeRnR.sequence.status.currentStep, in2 := #JOB_5_STEP_01)
      Contact( "Unit1.Em5.ControlNodes".gaugeRnR.sequence.status.seqActive )
      wire#w1
      Coil( "Unit1.Em5.ControlNodes".gaugeRnR."step".action1[501] )
   END_RUNG
   RUNG wire#w1
      Coil( "Unit1.Em5.ControlNodes".gaugeRnR."step".transition1[501] )
   END_RUNG
   RUNG wire#w1
      Contact( "Unit1.Em5.ControlNodes".gaugeRnR."step".transition1[501] )
      Move(in := #JOB_5_STEP_90, out1 => "Unit1.Em5.ControlNodes".gaugeRnR.sequence.status.nextStep)
   END_RUNG
   // the same network as SCL:
   "Unit1.Em5.ControlNodes".gaugeRnR."step".action1[501] := ("Unit1.Em5.ControlNodes".gaugeRnR.sequence.status.currentStep = #JOB_5_STEP_01) AND "Unit1.Em5.ControlNodes".gaugeRnR.sequence.status.seqActive;
   "Unit1.Em5.ControlNodes".gaugeRnR."step".transition1[501] := ("Unit1.Em5.ControlNodes".gaugeRnR.sequence.status.currentStep = #JOB_5_STEP_01) AND "Unit1.Em5.ControlNodes".gaugeRnR.sequence.status.seqActive;
   IF ("Unit1.Em5.ControlNodes".gaugeRnR.sequence.status.currentStep = #JOB_5_STEP_01) AND "Unit1.Em5.ControlNodes".gaugeRnR.sequence.status.seqActive AND "Unit1.Em5.ControlNodes".gaugeRnR."step".transition1[501] THEN
       "Unit1.Em5.ControlNodes".gaugeRnR.sequence.status.nextStep := #JOB_5_STEP_90;
   END_IF;
END_REGION

REGION Network 35: Step[510] : MainPnP1 X-Axis Move ReelCut Convyeor
   RUNG wire#powerrail
      { S7_Templates := "SrcType := DInt" } EQ_Contact(in1 := "Unit1.Em5.ControlNodes".gaugeRnR.sequence.status.currentStep, in2 := #JOB_5_STEP_10)
      Contact( "Unit1.Em5.ControlNodes".gaugeRnR.sequence.status.seqActive )
      wire#w1
      Coil( "Unit1.Em5.ControlNodes".gaugeRnR."step".action1[510] )
   END_RUNG
   RUNG wire#w1
      Contact( "Unit1.Em5.ControlNodes".cm.softCam.cathodeMainPnP1AxisX.reelCutConveyerPos.inPos )
      Coil( "Unit1.Em5.ControlNodes".gaugeRnR."step".transition1[510] )
   END_RUNG
   RUNG wire#w1
      Contact( "Unit1.Em5.ControlNodes".gaugeRnR."step".transition1[510] )
      Move(in := #JOB_5_STEP_20, out1 => "Unit1.Em5.ControlNodes".gaugeRnR.sequence.status.nextStep)
   END_RUNG
   // the same network as SCL:
   "Unit1.Em5.ControlNodes".gaugeRnR."step".action1[510] := ("Unit1.Em5.ControlNodes".gaugeRnR.sequence.status.currentStep = #JOB_5_STEP_10) AND "Unit1.Em5.ControlNodes".gaugeRnR.sequence.status.seqActive;
   "Unit1.Em5.ControlNodes".gaugeRnR."step".transition1[510] := ("Unit1.Em5.ControlNodes".gaugeRnR.sequence.status.currentStep = #JOB_5_STEP_10) AND "Unit1.Em5.ControlNodes".gaugeRnR.sequence.status.seqActive AND "Unit1.Em5.ControlNodes".cm.softCam.cathodeMainPnP1AxisX.reelCutConveyerPos.inPos;
   IF ("Unit1.Em5.ControlNodes".gaugeRnR.sequence.status.currentStep = #JOB_5_STEP_10) AND "Unit1.Em5.ControlNodes".gaugeRnR.sequence.status.seqActive AND "Unit1.Em5.ControlNodes".gaugeRnR."step".transition1[510] THEN
       "Unit1.Em5.ControlNodes".gaugeRnR.sequence.status.nextStep := #JOB_5_STEP_20;
   END_IF;
END_REGION

REGION Network 36: Step[520] : MainPnP2 X-Axis Move AlignTable
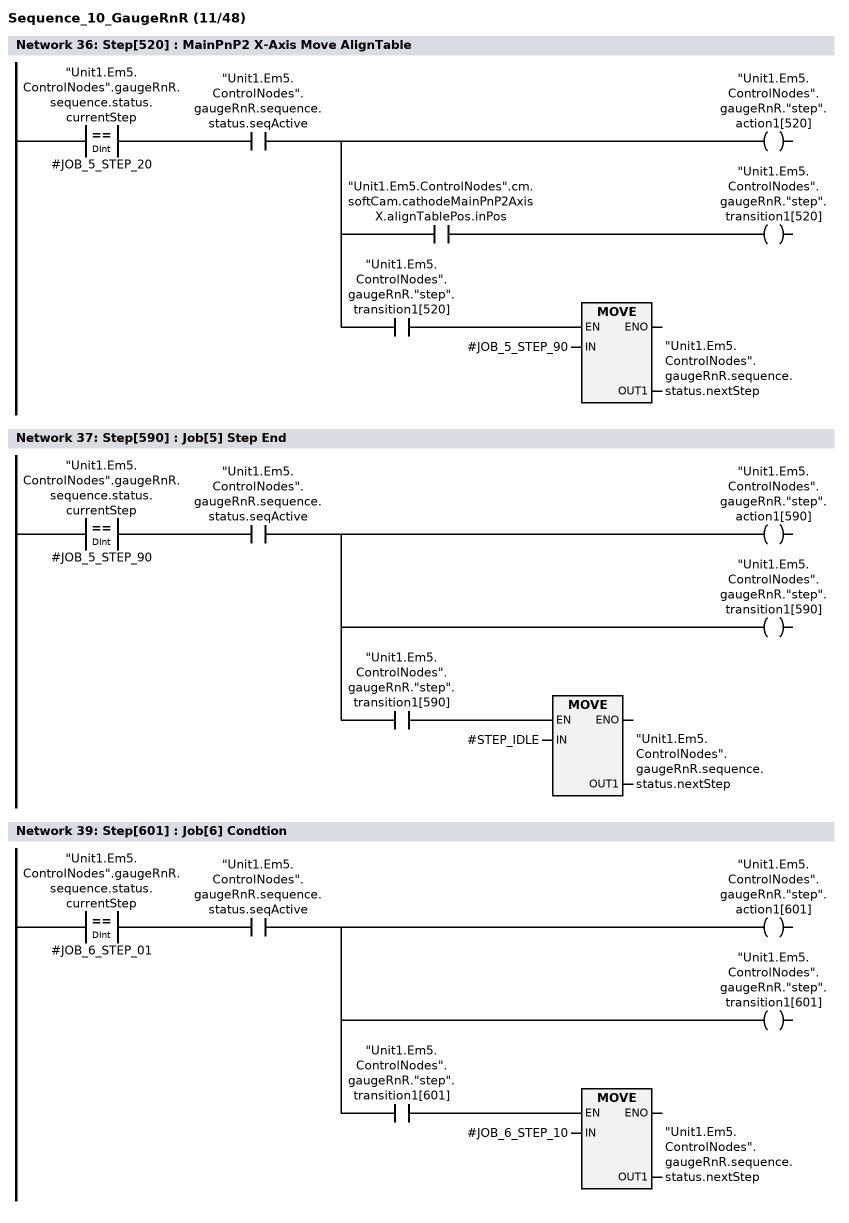
   RUNG wire#powerrail
      { S7_Templates := "SrcType := DInt" } EQ_Contact(in1 := "Unit1.Em5.ControlNodes".gaugeRnR.sequence.status.currentStep, in2 := #JOB_5_STEP_20)
      Contact( "Unit1.Em5.ControlNodes".gaugeRnR.sequence.status.seqActive )
      wire#w1
      Coil( "Unit1.Em5.ControlNodes".gaugeRnR."step".action1[520] )
   END_RUNG
   RUNG wire#w1
      Contact( "Unit1.Em5.ControlNodes".cm.softCam.cathodeMainPnP2AxisX.alignTablePos.inPos )
      Coil( "Unit1.Em5.ControlNodes".gaugeRnR."step".transition1[520] )
   END_RUNG
   RUNG wire#w1
      Contact( "Unit1.Em5.ControlNodes".gaugeRnR."step".transition1[520] )
      Move(in := #JOB_5_STEP_90, out1 => "Unit1.Em5.ControlNodes".gaugeRnR.sequence.status.nextStep)
   END_RUNG
   // the same network as SCL:
   "Unit1.Em5.ControlNodes".gaugeRnR."step".action1[520] := ("Unit1.Em5.ControlNodes".gaugeRnR.sequence.status.currentStep = #JOB_5_STEP_20) AND "Unit1.Em5.ControlNodes".gaugeRnR.sequence.status.seqActive;
   "Unit1.Em5.ControlNodes".gaugeRnR."step".transition1[520] := ("Unit1.Em5.ControlNodes".gaugeRnR.sequence.status.currentStep = #JOB_5_STEP_20) AND "Unit1.Em5.ControlNodes".gaugeRnR.sequence.status.seqActive AND "Unit1.Em5.ControlNodes".cm.softCam.cathodeMainPnP2AxisX.alignTablePos.inPos;
   IF ("Unit1.Em5.ControlNodes".gaugeRnR.sequence.status.currentStep = #JOB_5_STEP_20) AND "Unit1.Em5.ControlNodes".gaugeRnR.sequence.status.seqActive AND "Unit1.Em5.ControlNodes".gaugeRnR."step".transition1[520] THEN
       "Unit1.Em5.ControlNodes".gaugeRnR.sequence.status.nextStep := #JOB_5_STEP_90;
   END_IF;
END_REGION

REGION Network 37: Step[590] : Job[5] Step End
   RUNG wire#powerrail
      { S7_Templates := "SrcType := DInt" } EQ_Contact(in1 := "Unit1.Em5.ControlNodes".gaugeRnR.sequence.status.currentStep, in2 := #JOB_5_STEP_90)
      Contact( "Unit1.Em5.ControlNodes".gaugeRnR.sequence.status.seqActive )
      wire#w1
      Coil( "Unit1.Em5.ControlNodes".gaugeRnR."step".action1[590] )
   END_RUNG
   RUNG wire#w1
      Coil( "Unit1.Em5.ControlNodes".gaugeRnR."step".transition1[590] )
   END_RUNG
   RUNG wire#w1
      Contact( "Unit1.Em5.ControlNodes".gaugeRnR."step".transition1[590] )
      Move(in := #STEP_IDLE, out1 => "Unit1.Em5.ControlNodes".gaugeRnR.sequence.status.nextStep)
   END_RUNG
   // the same network as SCL:
   "Unit1.Em5.ControlNodes".gaugeRnR."step".action1[590] := ("Unit1.Em5.ControlNodes".gaugeRnR.sequence.status.currentStep = #JOB_5_STEP_90) AND "Unit1.Em5.ControlNodes".gaugeRnR.sequence.status.seqActive;
   "Unit1.Em5.ControlNodes".gaugeRnR."step".transition1[590] := ("Unit1.Em5.ControlNodes".gaugeRnR.sequence.status.currentStep = #JOB_5_STEP_90) AND "Unit1.Em5.ControlNodes".gaugeRnR.sequence.status.seqActive;
   IF ("Unit1.Em5.ControlNodes".gaugeRnR.sequence.status.currentStep = #JOB_5_STEP_90) AND "Unit1.Em5.ControlNodes".gaugeRnR.sequence.status.seqActive AND "Unit1.Em5.ControlNodes".gaugeRnR."step".transition1[590] THEN
       "Unit1.Em5.ControlNodes".gaugeRnR.sequence.status.nextStep := #STEP_IDLE;
   END_IF;
END_REGION

REGION Network 38: *************** JOB[6] Common AlignTable Vision Adjust ************************
END_REGION

REGION Network 39: Step[601] : Job[6] Condtion
   RUNG wire#powerrail
      { S7_Templates := "SrcType := DInt" } EQ_Contact(in1 := "Unit1.Em5.ControlNodes".gaugeRnR.sequence.status.currentStep, in2 := #JOB_6_STEP_01)
      Contact( "Unit1.Em5.ControlNodes".gaugeRnR.sequence.status.seqActive )
      wire#w1
      Coil( "Unit1.Em5.ControlNodes".gaugeRnR."step".action1[601] )
   END_RUNG
   RUNG wire#w1
      Coil( "Unit1.Em5.ControlNodes".gaugeRnR."step".transition1[601] )
   END_RUNG
   RUNG wire#w1
      Contact( "Unit1.Em5.ControlNodes".gaugeRnR."step".transition1[601] )
      Move(in := #JOB_6_STEP_10, out1 => "Unit1.Em5.ControlNodes".gaugeRnR.sequence.status.nextStep)
   END_RUNG
   // the same network as SCL:
   "Unit1.Em5.ControlNodes".gaugeRnR."step".action1[601] := ("Unit1.Em5.ControlNodes".gaugeRnR.sequence.status.currentStep = #JOB_6_STEP_01) AND "Unit1.Em5.ControlNodes".gaugeRnR.sequence.status.seqActive;
   "Unit1.Em5.ControlNodes".gaugeRnR."step".transition1[601] := ("Unit1.Em5.ControlNodes".gaugeRnR.sequence.status.currentStep = #JOB_6_STEP_01) AND "Unit1.Em5.ControlNodes".gaugeRnR.sequence.status.seqActive;
   IF ("Unit1.Em5.ControlNodes".gaugeRnR.sequence.status.currentStep = #JOB_6_STEP_01) AND "Unit1.Em5.ControlNodes".gaugeRnR.sequence.status.seqActive AND "Unit1.Em5.ControlNodes".gaugeRnR."step".transition1[601] THEN
       "Unit1.Em5.ControlNodes".gaugeRnR.sequence.status.nextStep := #JOB_6_STEP_10;
   END_IF;
END_REGION

REGION Network 40: Step[610] : AlignTable Vision Trigger On
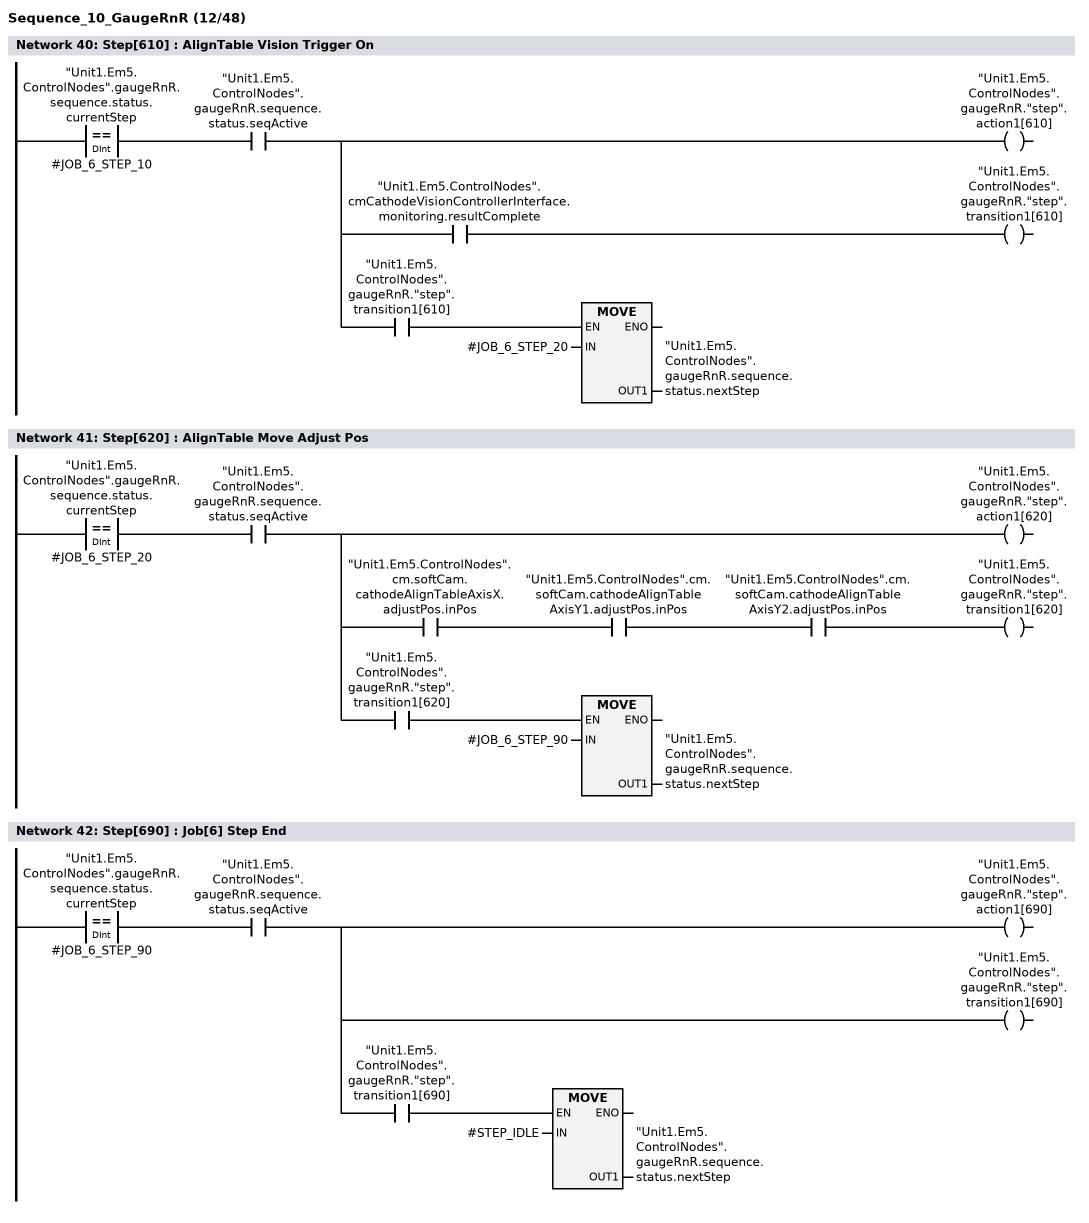
   RUNG wire#powerrail
      { S7_Templates := "SrcType := DInt" } EQ_Contact(in1 := "Unit1.Em5.ControlNodes".gaugeRnR.sequence.status.currentStep, in2 := #JOB_6_STEP_10)
      Contact( "Unit1.Em5.ControlNodes".gaugeRnR.sequence.status.seqActive )
      wire#w1
      Coil( "Unit1.Em5.ControlNodes".gaugeRnR."step".action1[610] )
   END_RUNG
   RUNG wire#w1
      Contact( "Unit1.Em5.ControlNodes".cmCathodeVisionControllerInterface.monitoring.resultComplete )
      Coil( "Unit1.Em5.ControlNodes".gaugeRnR."step".transition1[610] )
   END_RUNG
   RUNG wire#w1
      Contact( "Unit1.Em5.ControlNodes".gaugeRnR."step".transition1[610] )
      Move(in := #JOB_6_STEP_20, out1 => "Unit1.Em5.ControlNodes".gaugeRnR.sequence.status.nextStep)
   END_RUNG
   // the same network as SCL:
   "Unit1.Em5.ControlNodes".gaugeRnR."step".action1[610] := ("Unit1.Em5.ControlNodes".gaugeRnR.sequence.status.currentStep = #JOB_6_STEP_10) AND "Unit1.Em5.ControlNodes".gaugeRnR.sequence.status.seqActive;
   "Unit1.Em5.ControlNodes".gaugeRnR."step".transition1[610] := ("Unit1.Em5.ControlNodes".gaugeRnR.sequence.status.currentStep = #JOB_6_STEP_10) AND "Unit1.Em5.ControlNodes".gaugeRnR.sequence.status.seqActive AND "Unit1.Em5.ControlNodes".cmCathodeVisionControllerInterface.monitoring.resultComplete;
   IF ("Unit1.Em5.ControlNodes".gaugeRnR.sequence.status.currentStep = #JOB_6_STEP_10) AND "Unit1.Em5.ControlNodes".gaugeRnR.sequence.status.seqActive AND "Unit1.Em5.ControlNodes".gaugeRnR."step".transition1[610] THEN
       "Unit1.Em5.ControlNodes".gaugeRnR.sequence.status.nextStep := #JOB_6_STEP_20;
   END_IF;
END_REGION

REGION Network 41: Step[620] : AlignTable Move Adjust Pos
   RUNG wire#powerrail
      { S7_Templates := "SrcType := DInt" } EQ_Contact(in1 := "Unit1.Em5.ControlNodes".gaugeRnR.sequence.status.currentStep, in2 := #JOB_6_STEP_20)
      Contact( "Unit1.Em5.ControlNodes".gaugeRnR.sequence.status.seqActive )
      wire#w1
      Coil( "Unit1.Em5.ControlNodes".gaugeRnR."step".action1[620] )
   END_RUNG
   RUNG wire#w1
      Contact( "Unit1.Em5.ControlNodes".cm.softCam.cathodeAlignTableAxisX.adjustPos.inPos )
      Contact( "Unit1.Em5.ControlNodes".cm.softCam.cathodeAlignTableAxisY1.adjustPos.inPos )
      Contact( "Unit1.Em5.ControlNodes".cm.softCam.cathodeAlignTableAxisY2.adjustPos.inPos )
      Coil( "Unit1.Em5.ControlNodes".gaugeRnR."step".transition1[620] )
   END_RUNG
   RUNG wire#w1
      Contact( "Unit1.Em5.ControlNodes".gaugeRnR."step".transition1[620] )
      Move(in := #JOB_6_STEP_90, out1 => "Unit1.Em5.ControlNodes".gaugeRnR.sequence.status.nextStep)
   END_RUNG
   // the same network as SCL:
   "Unit1.Em5.ControlNodes".gaugeRnR."step".action1[620] := ("Unit1.Em5.ControlNodes".gaugeRnR.sequence.status.currentStep = #JOB_6_STEP_20) AND "Unit1.Em5.ControlNodes".gaugeRnR.sequence.status.seqActive;
   "Unit1.Em5.ControlNodes".gaugeRnR."step".transition1[620] := ("Unit1.Em5.ControlNodes".gaugeRnR.sequence.status.currentStep = #JOB_6_STEP_20) AND "Unit1.Em5.ControlNodes".gaugeRnR.sequence.status.seqActive AND "Unit1.Em5.ControlNodes".cm.softCam.cathodeAlignTableAxisX.adjustPos.inPos AND "Unit1.Em5.ControlNodes".cm.softCam.cathodeAlignTableAxisY1.adjustPos.inPos AND "Unit1.Em5.ControlNodes".cm.softCam.cathodeAlignTableAxisY2.adjustPos.inPos;
   IF ("Unit1.Em5.ControlNodes".gaugeRnR.sequence.status.currentStep = #JOB_6_STEP_20) AND "Unit1.Em5.ControlNodes".gaugeRnR.sequence.status.seqActive AND "Unit1.Em5.ControlNodes".gaugeRnR."step".transition1[620] THEN
       "Unit1.Em5.ControlNodes".gaugeRnR.sequence.status.nextStep := #JOB_6_STEP_90;
   END_IF;
END_REGION

REGION Network 42: Step[690] : Job[6] Step End
   RUNG wire#powerrail
      { S7_Templates := "SrcType := DInt" } EQ_Contact(in1 := "Unit1.Em5.ControlNodes".gaugeRnR.sequence.status.currentStep, in2 := #JOB_6_STEP_90)
      Contact( "Unit1.Em5.ControlNodes".gaugeRnR.sequence.status.seqActive )
      wire#w1
      Coil( "Unit1.Em5.ControlNodes".gaugeRnR."step".action1[690] )
   END_RUNG
   RUNG wire#w1
      Coil( "Unit1.Em5.ControlNodes".gaugeRnR."step".transition1[690] )
   END_RUNG
   RUNG wire#w1
      Contact( "Unit1.Em5.ControlNodes".gaugeRnR."step".transition1[690] )
      Move(in := #STEP_IDLE, out1 => "Unit1.Em5.ControlNodes".gaugeRnR.sequence.status.nextStep)
   END_RUNG
   // the same network as SCL:
   "Unit1.Em5.ControlNodes".gaugeRnR."step".action1[690] := ("Unit1.Em5.ControlNodes".gaugeRnR.sequence.status.currentStep = #JOB_6_STEP_90) AND "Unit1.Em5.ControlNodes".gaugeRnR.sequence.status.seqActive;
   "Unit1.Em5.ControlNodes".gaugeRnR."step".transition1[690] := ("Unit1.Em5.ControlNodes".gaugeRnR.sequence.status.currentStep = #JOB_6_STEP_90) AND "Unit1.Em5.ControlNodes".gaugeRnR.sequence.status.seqActive;
   IF ("Unit1.Em5.ControlNodes".gaugeRnR.sequence.status.currentStep = #JOB_6_STEP_90) AND "Unit1.Em5.ControlNodes".gaugeRnR.sequence.status.seqActive AND "Unit1.Em5.ControlNodes".gaugeRnR."step".transition1[690] THEN
       "Unit1.Em5.ControlNodes".gaugeRnR.sequence.status.nextStep := #STEP_IDLE;
   END_IF;
END_REGION

REGION Network 43: *************** JOB[10] AlignTable To MainPnP1 ************************
END_REGION

REGION Network 44: Step[1001] : Job[10] Condtion
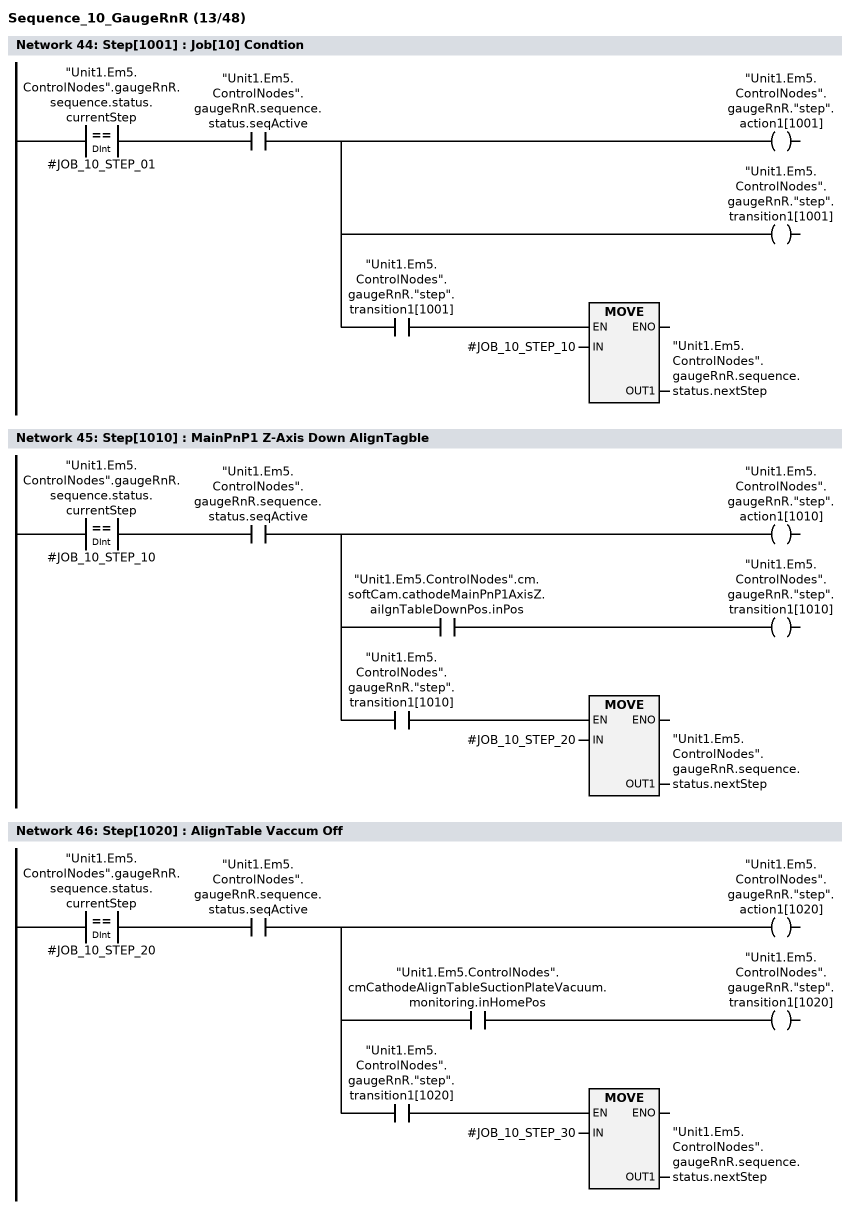
   RUNG wire#powerrail
      { S7_Templates := "SrcType := DInt" } EQ_Contact(in1 := "Unit1.Em5.ControlNodes".gaugeRnR.sequence.status.currentStep, in2 := #JOB_10_STEP_01)
      Contact( "Unit1.Em5.ControlNodes".gaugeRnR.sequence.status.seqActive )
      wire#w1
      Coil( "Unit1.Em5.ControlNodes".gaugeRnR."step".action1[1001] )
   END_RUNG
   RUNG wire#w1
      Coil( "Unit1.Em5.ControlNodes".gaugeRnR."step".transition1[1001] )
   END_RUNG
   RUNG wire#w1
      Contact( "Unit1.Em5.ControlNodes".gaugeRnR."step".transition1[1001] )
      Move(in := #JOB_10_STEP_10, out1 => "Unit1.Em5.ControlNodes".gaugeRnR.sequence.status.nextStep)
   END_RUNG
   // the same network as SCL:
   "Unit1.Em5.ControlNodes".gaugeRnR."step".action1[1001] := ("Unit1.Em5.ControlNodes".gaugeRnR.sequence.status.currentStep = #JOB_10_STEP_01) AND "Unit1.Em5.ControlNodes".gaugeRnR.sequence.status.seqActive;
   "Unit1.Em5.ControlNodes".gaugeRnR."step".transition1[1001] := ("Unit1.Em5.ControlNodes".gaugeRnR.sequence.status.currentStep = #JOB_10_STEP_01) AND "Unit1.Em5.ControlNodes".gaugeRnR.sequence.status.seqActive;
   IF ("Unit1.Em5.ControlNodes".gaugeRnR.sequence.status.currentStep = #JOB_10_STEP_01) AND "Unit1.Em5.ControlNodes".gaugeRnR.sequence.status.seqActive AND "Unit1.Em5.ControlNodes".gaugeRnR."step".transition1[1001] THEN
       "Unit1.Em5.ControlNodes".gaugeRnR.sequence.status.nextStep := #JOB_10_STEP_10;
   END_IF;
END_REGION

REGION Network 45: Step[1010] : MainPnP1 Z-Axis Down AlignTagble
   RUNG wire#powerrail
      { S7_Templates := "SrcType := DInt" } EQ_Contact(in1 := "Unit1.Em5.ControlNodes".gaugeRnR.sequence.status.currentStep, in2 := #JOB_10_STEP_10)
      Contact( "Unit1.Em5.ControlNodes".gaugeRnR.sequence.status.seqActive )
      wire#w1
      Coil( "Unit1.Em5.ControlNodes".gaugeRnR."step".action1[1010] )
   END_RUNG
   RUNG wire#w1
      Contact( "Unit1.Em5.ControlNodes".cm.softCam.cathodeMainPnP1AxisZ.ailgnTableDownPos.inPos )
      Coil( "Unit1.Em5.ControlNodes".gaugeRnR."step".transition1[1010] )
   END_RUNG
   RUNG wire#w1
      Contact( "Unit1.Em5.ControlNodes".gaugeRnR."step".transition1[1010] )
      Move(in := #JOB_10_STEP_20, out1 => "Unit1.Em5.ControlNodes".gaugeRnR.sequence.status.nextStep)
   END_RUNG
   // the same network as SCL:
   "Unit1.Em5.ControlNodes".gaugeRnR."step".action1[1010] := ("Unit1.Em5.ControlNodes".gaugeRnR.sequence.status.currentStep = #JOB_10_STEP_10) AND "Unit1.Em5.ControlNodes".gaugeRnR.sequence.status.seqActive;
   "Unit1.Em5.ControlNodes".gaugeRnR."step".transition1[1010] := ("Unit1.Em5.ControlNodes".gaugeRnR.sequence.status.currentStep = #JOB_10_STEP_10) AND "Unit1.Em5.ControlNodes".gaugeRnR.sequence.status.seqActive AND "Unit1.Em5.ControlNodes".cm.softCam.cathodeMainPnP1AxisZ.ailgnTableDownPos.inPos;
   IF ("Unit1.Em5.ControlNodes".gaugeRnR.sequence.status.currentStep = #JOB_10_STEP_10) AND "Unit1.Em5.ControlNodes".gaugeRnR.sequence.status.seqActive AND "Unit1.Em5.ControlNodes".gaugeRnR."step".transition1[1010] THEN
       "Unit1.Em5.ControlNodes".gaugeRnR.sequence.status.nextStep := #JOB_10_STEP_20;
   END_IF;
END_REGION

REGION Network 46: Step[1020] : AlignTable Vaccum Off
   RUNG wire#powerrail
      { S7_Templates := "SrcType := DInt" } EQ_Contact(in1 := "Unit1.Em5.ControlNodes".gaugeRnR.sequence.status.currentStep, in2 := #JOB_10_STEP_20)
      Contact( "Unit1.Em5.ControlNodes".gaugeRnR.sequence.status.seqActive )
      wire#w1
      Coil( "Unit1.Em5.ControlNodes".gaugeRnR."step".action1[1020] )
   END_RUNG
   RUNG wire#w1
      Contact( "Unit1.Em5.ControlNodes".cmCathodeAlignTableSuctionPlateVacuum.monitoring.inHomePos )
      Coil( "Unit1.Em5.ControlNodes".gaugeRnR."step".transition1[1020] )
   END_RUNG
   RUNG wire#w1
      Contact( "Unit1.Em5.ControlNodes".gaugeRnR."step".transition1[1020] )
      Move(in := #JOB_10_STEP_30, out1 => "Unit1.Em5.ControlNodes".gaugeRnR.sequence.status.nextStep)
   END_RUNG
   // the same network as SCL:
   "Unit1.Em5.ControlNodes".gaugeRnR."step".action1[1020] := ("Unit1.Em5.ControlNodes".gaugeRnR.sequence.status.currentStep = #JOB_10_STEP_20) AND "Unit1.Em5.ControlNodes".gaugeRnR.sequence.status.seqActive;
   "Unit1.Em5.ControlNodes".gaugeRnR."step".transition1[1020] := ("Unit1.Em5.ControlNodes".gaugeRnR.sequence.status.currentStep = #JOB_10_STEP_20) AND "Unit1.Em5.ControlNodes".gaugeRnR.sequence.status.seqActive AND "Unit1.Em5.ControlNodes".cmCathodeAlignTableSuctionPlateVacuum.monitoring.inHomePos;
   IF ("Unit1.Em5.ControlNodes".gaugeRnR.sequence.status.currentStep = #JOB_10_STEP_20) AND "Unit1.Em5.ControlNodes".gaugeRnR.sequence.status.seqActive AND "Unit1.Em5.ControlNodes".gaugeRnR."step".transition1[1020] THEN
       "Unit1.Em5.ControlNodes".gaugeRnR.sequence.status.nextStep := #JOB_10_STEP_30;
   END_IF;
END_REGION

REGION Network 47: Step[1030] : MainPnP1 Vaccum On
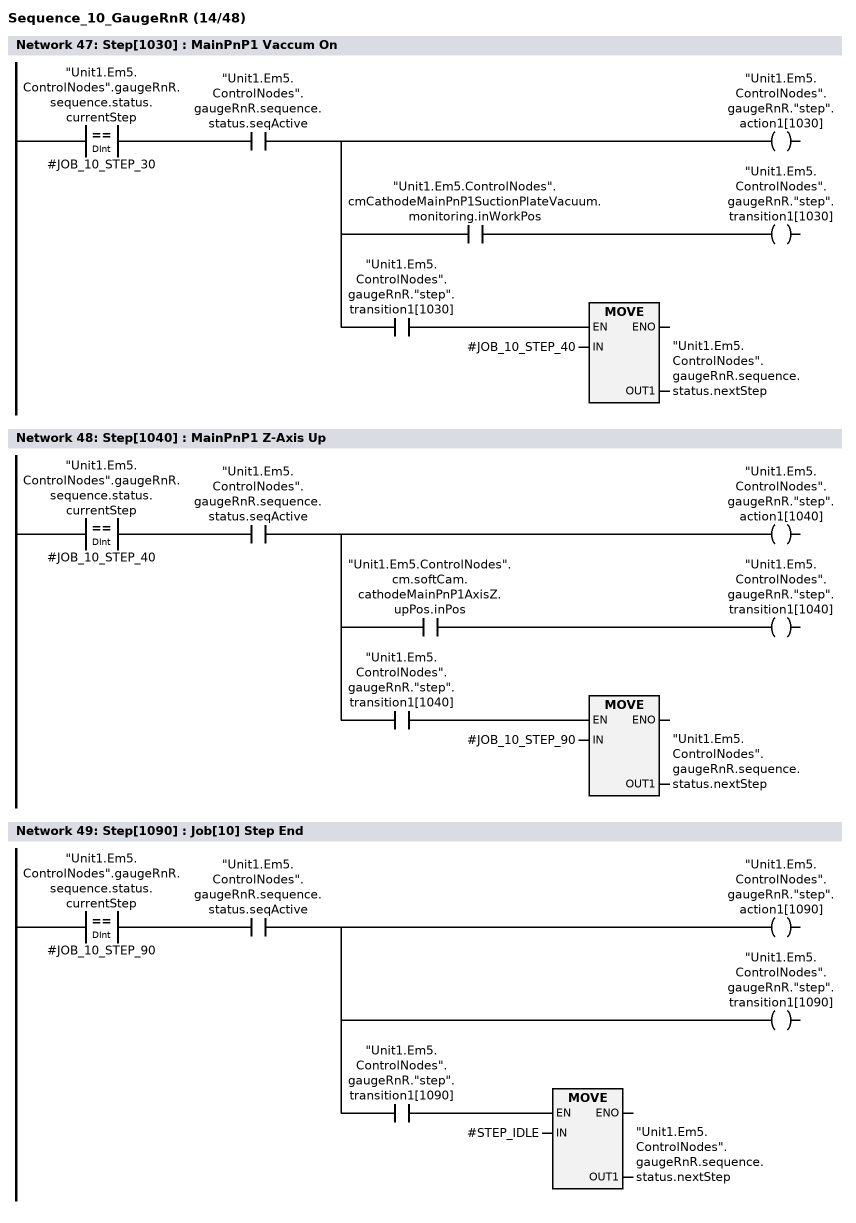
   RUNG wire#powerrail
      { S7_Templates := "SrcType := DInt" } EQ_Contact(in1 := "Unit1.Em5.ControlNodes".gaugeRnR.sequence.status.currentStep, in2 := #JOB_10_STEP_30)
      Contact( "Unit1.Em5.ControlNodes".gaugeRnR.sequence.status.seqActive )
      wire#w1
      Coil( "Unit1.Em5.ControlNodes".gaugeRnR."step".action1[1030] )
   END_RUNG
   RUNG wire#w1
      Contact( "Unit1.Em5.ControlNodes".cmCathodeMainPnP1SuctionPlateVacuum.monitoring.inWorkPos )
      Coil( "Unit1.Em5.ControlNodes".gaugeRnR."step".transition1[1030] )
   END_RUNG
   RUNG wire#w1
      Contact( "Unit1.Em5.ControlNodes".gaugeRnR."step".transition1[1030] )
      Move(in := #JOB_10_STEP_40, out1 => "Unit1.Em5.ControlNodes".gaugeRnR.sequence.status.nextStep)
   END_RUNG
   // the same network as SCL:
   "Unit1.Em5.ControlNodes".gaugeRnR."step".action1[1030] := ("Unit1.Em5.ControlNodes".gaugeRnR.sequence.status.currentStep = #JOB_10_STEP_30) AND "Unit1.Em5.ControlNodes".gaugeRnR.sequence.status.seqActive;
   "Unit1.Em5.ControlNodes".gaugeRnR."step".transition1[1030] := ("Unit1.Em5.ControlNodes".gaugeRnR.sequence.status.currentStep = #JOB_10_STEP_30) AND "Unit1.Em5.ControlNodes".gaugeRnR.sequence.status.seqActive AND "Unit1.Em5.ControlNodes".cmCathodeMainPnP1SuctionPlateVacuum.monitoring.inWorkPos;
   IF ("Unit1.Em5.ControlNodes".gaugeRnR.sequence.status.currentStep = #JOB_10_STEP_30) AND "Unit1.Em5.ControlNodes".gaugeRnR.sequence.status.seqActive AND "Unit1.Em5.ControlNodes".gaugeRnR."step".transition1[1030] THEN
       "Unit1.Em5.ControlNodes".gaugeRnR.sequence.status.nextStep := #JOB_10_STEP_40;
   END_IF;
END_REGION

REGION Network 48: Step[1040] : MainPnP1 Z-Axis Up
   RUNG wire#powerrail
      { S7_Templates := "SrcType := DInt" } EQ_Contact(in1 := "Unit1.Em5.ControlNodes".gaugeRnR.sequence.status.currentStep, in2 := #JOB_10_STEP_40)
      Contact( "Unit1.Em5.ControlNodes".gaugeRnR.sequence.status.seqActive )
      wire#w1
      Coil( "Unit1.Em5.ControlNodes".gaugeRnR."step".action1[1040] )
   END_RUNG
   RUNG wire#w1
      Contact( "Unit1.Em5.ControlNodes".cm.softCam.cathodeMainPnP1AxisZ.upPos.inPos )
      Coil( "Unit1.Em5.ControlNodes".gaugeRnR."step".transition1[1040] )
   END_RUNG
   RUNG wire#w1
      Contact( "Unit1.Em5.ControlNodes".gaugeRnR."step".transition1[1040] )
      Move(in := #JOB_10_STEP_90, out1 => "Unit1.Em5.ControlNodes".gaugeRnR.sequence.status.nextStep)
   END_RUNG
   // the same network as SCL:
   "Unit1.Em5.ControlNodes".gaugeRnR."step".action1[1040] := ("Unit1.Em5.ControlNodes".gaugeRnR.sequence.status.currentStep = #JOB_10_STEP_40) AND "Unit1.Em5.ControlNodes".gaugeRnR.sequence.status.seqActive;
   "Unit1.Em5.ControlNodes".gaugeRnR."step".transition1[1040] := ("Unit1.Em5.ControlNodes".gaugeRnR.sequence.status.currentStep = #JOB_10_STEP_40) AND "Unit1.Em5.ControlNodes".gaugeRnR.sequence.status.seqActive AND "Unit1.Em5.ControlNodes".cm.softCam.cathodeMainPnP1AxisZ.upPos.inPos;
   IF ("Unit1.Em5.ControlNodes".gaugeRnR.sequence.status.currentStep = #JOB_10_STEP_40) AND "Unit1.Em5.ControlNodes".gaugeRnR.sequence.status.seqActive AND "Unit1.Em5.ControlNodes".gaugeRnR."step".transition1[1040] THEN
       "Unit1.Em5.ControlNodes".gaugeRnR.sequence.status.nextStep := #JOB_10_STEP_90;
   END_IF;
END_REGION

REGION Network 49: Step[1090] : Job[10] Step End
   RUNG wire#powerrail
      { S7_Templates := "SrcType := DInt" } EQ_Contact(in1 := "Unit1.Em5.ControlNodes".gaugeRnR.sequence.status.currentStep, in2 := #JOB_10_STEP_90)
      Contact( "Unit1.Em5.ControlNodes".gaugeRnR.sequence.status.seqActive )
      wire#w1
      Coil( "Unit1.Em5.ControlNodes".gaugeRnR."step".action1[1090] )
   END_RUNG
   RUNG wire#w1
      Coil( "Unit1.Em5.ControlNodes".gaugeRnR."step".transition1[1090] )
   END_RUNG
   RUNG wire#w1
      Contact( "Unit1.Em5.ControlNodes".gaugeRnR."step".transition1[1090] )
      Move(in := #STEP_IDLE, out1 => "Unit1.Em5.ControlNodes".gaugeRnR.sequence.status.nextStep)
   END_RUNG
   // the same network as SCL:
   "Unit1.Em5.ControlNodes".gaugeRnR."step".action1[1090] := ("Unit1.Em5.ControlNodes".gaugeRnR.sequence.status.currentStep = #JOB_10_STEP_90) AND "Unit1.Em5.ControlNodes".gaugeRnR.sequence.status.seqActive;
   "Unit1.Em5.ControlNodes".gaugeRnR."step".transition1[1090] := ("Unit1.Em5.ControlNodes".gaugeRnR.sequence.status.currentStep = #JOB_10_STEP_90) AND "Unit1.Em5.ControlNodes".gaugeRnR.sequence.status.seqActive;
   IF ("Unit1.Em5.ControlNodes".gaugeRnR.sequence.status.currentStep = #JOB_10_STEP_90) AND "Unit1.Em5.ControlNodes".gaugeRnR.sequence.status.seqActive AND "Unit1.Em5.ControlNodes".gaugeRnR."step".transition1[1090] THEN
       "Unit1.Em5.ControlNodes".gaugeRnR.sequence.status.nextStep := #STEP_IDLE;
   END_IF;
END_REGION

REGION Network 50: *************** JOB[11] MainPnP Move ReelCut Convyeor / AlignTable************************
END_REGION

REGION Network 51: Step[1101] : Job[11] Condtion
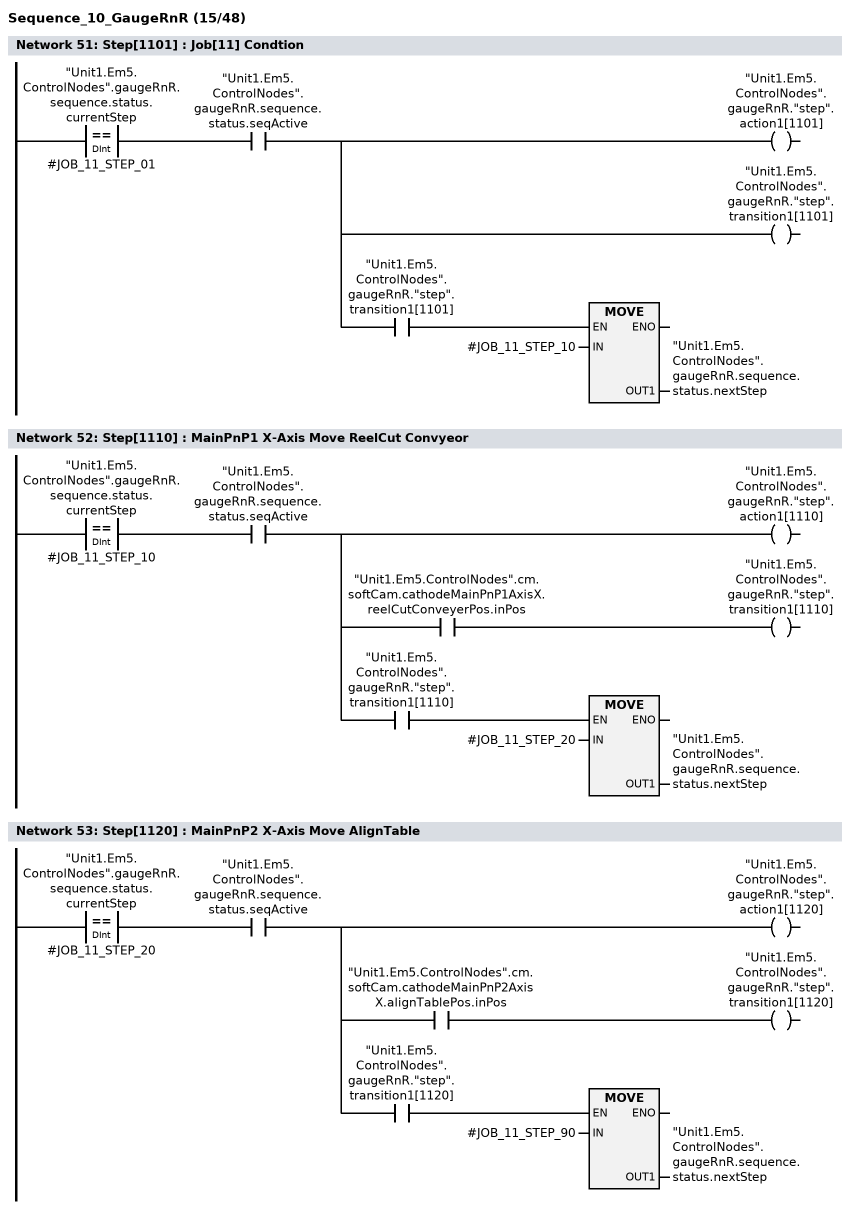
   RUNG wire#powerrail
      { S7_Templates := "SrcType := DInt" } EQ_Contact(in1 := "Unit1.Em5.ControlNodes".gaugeRnR.sequence.status.currentStep, in2 := #JOB_11_STEP_01)
      Contact( "Unit1.Em5.ControlNodes".gaugeRnR.sequence.status.seqActive )
      wire#w1
      Coil( "Unit1.Em5.ControlNodes".gaugeRnR."step".action1[1101] )
   END_RUNG
   RUNG wire#w1
      Coil( "Unit1.Em5.ControlNodes".gaugeRnR."step".transition1[1101] )
   END_RUNG
   RUNG wire#w1
      Contact( "Unit1.Em5.ControlNodes".gaugeRnR."step".transition1[1101] )
      Move(in := #JOB_11_STEP_10, out1 => "Unit1.Em5.ControlNodes".gaugeRnR.sequence.status.nextStep)
   END_RUNG
   // the same network as SCL:
   "Unit1.Em5.ControlNodes".gaugeRnR."step".action1[1101] := ("Unit1.Em5.ControlNodes".gaugeRnR.sequence.status.currentStep = #JOB_11_STEP_01) AND "Unit1.Em5.ControlNodes".gaugeRnR.sequence.status.seqActive;
   "Unit1.Em5.ControlNodes".gaugeRnR."step".transition1[1101] := ("Unit1.Em5.ControlNodes".gaugeRnR.sequence.status.currentStep = #JOB_11_STEP_01) AND "Unit1.Em5.ControlNodes".gaugeRnR.sequence.status.seqActive;
   IF ("Unit1.Em5.ControlNodes".gaugeRnR.sequence.status.currentStep = #JOB_11_STEP_01) AND "Unit1.Em5.ControlNodes".gaugeRnR.sequence.status.seqActive AND "Unit1.Em5.ControlNodes".gaugeRnR."step".transition1[1101] THEN
       "Unit1.Em5.ControlNodes".gaugeRnR.sequence.status.nextStep := #JOB_11_STEP_10;
   END_IF;
END_REGION

REGION Network 52: Step[1110] : MainPnP1 X-Axis Move ReelCut Convyeor
   RUNG wire#powerrail
      { S7_Templates := "SrcType := DInt" } EQ_Contact(in1 := "Unit1.Em5.ControlNodes".gaugeRnR.sequence.status.currentStep, in2 := #JOB_11_STEP_10)
      Contact( "Unit1.Em5.ControlNodes".gaugeRnR.sequence.status.seqActive )
      wire#w1
      Coil( "Unit1.Em5.ControlNodes".gaugeRnR."step".action1[1110] )
   END_RUNG
   RUNG wire#w1
      Contact( "Unit1.Em5.ControlNodes".cm.softCam.cathodeMainPnP1AxisX.reelCutConveyerPos.inPos )
      Coil( "Unit1.Em5.ControlNodes".gaugeRnR."step".transition1[1110] )
   END_RUNG
   RUNG wire#w1
      Contact( "Unit1.Em5.ControlNodes".gaugeRnR."step".transition1[1110] )
      Move(in := #JOB_11_STEP_20, out1 => "Unit1.Em5.ControlNodes".gaugeRnR.sequence.status.nextStep)
   END_RUNG
   // the same network as SCL:
   "Unit1.Em5.ControlNodes".gaugeRnR."step".action1[1110] := ("Unit1.Em5.ControlNodes".gaugeRnR.sequence.status.currentStep = #JOB_11_STEP_10) AND "Unit1.Em5.ControlNodes".gaugeRnR.sequence.status.seqActive;
   "Unit1.Em5.ControlNodes".gaugeRnR."step".transition1[1110] := ("Unit1.Em5.ControlNodes".gaugeRnR.sequence.status.currentStep = #JOB_11_STEP_10) AND "Unit1.Em5.ControlNodes".gaugeRnR.sequence.status.seqActive AND "Unit1.Em5.ControlNodes".cm.softCam.cathodeMainPnP1AxisX.reelCutConveyerPos.inPos;
   IF ("Unit1.Em5.ControlNodes".gaugeRnR.sequence.status.currentStep = #JOB_11_STEP_10) AND "Unit1.Em5.ControlNodes".gaugeRnR.sequence.status.seqActive AND "Unit1.Em5.ControlNodes".gaugeRnR."step".transition1[1110] THEN
       "Unit1.Em5.ControlNodes".gaugeRnR.sequence.status.nextStep := #JOB_11_STEP_20;
   END_IF;
END_REGION

REGION Network 53: Step[1120] : MainPnP2 X-Axis Move AlignTable
   RUNG wire#powerrail
      { S7_Templates := "SrcType := DInt" } EQ_Contact(in1 := "Unit1.Em5.ControlNodes".gaugeRnR.sequence.status.currentStep, in2 := #JOB_11_STEP_20)
      Contact( "Unit1.Em5.ControlNodes".gaugeRnR.sequence.status.seqActive )
      wire#w1
      Coil( "Unit1.Em5.ControlNodes".gaugeRnR."step".action1[1120] )
   END_RUNG
   RUNG wire#w1
      Contact( "Unit1.Em5.ControlNodes".cm.softCam.cathodeMainPnP2AxisX.alignTablePos.inPos )
      Coil( "Unit1.Em5.ControlNodes".gaugeRnR."step".transition1[1120] )
   END_RUNG
   RUNG wire#w1
      Contact( "Unit1.Em5.ControlNodes".gaugeRnR."step".transition1[1120] )
      Move(in := #JOB_11_STEP_90, out1 => "Unit1.Em5.ControlNodes".gaugeRnR.sequence.status.nextStep)
   END_RUNG
   // the same network as SCL:
   "Unit1.Em5.ControlNodes".gaugeRnR."step".action1[1120] := ("Unit1.Em5.ControlNodes".gaugeRnR.sequence.status.currentStep = #JOB_11_STEP_20) AND "Unit1.Em5.ControlNodes".gaugeRnR.sequence.status.seqActive;
   "Unit1.Em5.ControlNodes".gaugeRnR."step".transition1[1120] := ("Unit1.Em5.ControlNodes".gaugeRnR.sequence.status.currentStep = #JOB_11_STEP_20) AND "Unit1.Em5.ControlNodes".gaugeRnR.sequence.status.seqActive AND "Unit1.Em5.ControlNodes".cm.softCam.cathodeMainPnP2AxisX.alignTablePos.inPos;
   IF ("Unit1.Em5.ControlNodes".gaugeRnR.sequence.status.currentStep = #JOB_11_STEP_20) AND "Unit1.Em5.ControlNodes".gaugeRnR.sequence.status.seqActive AND "Unit1.Em5.ControlNodes".gaugeRnR."step".transition1[1120] THEN
       "Unit1.Em5.ControlNodes".gaugeRnR.sequence.status.nextStep := #JOB_11_STEP_90;
   END_IF;
END_REGION

REGION Network 54: Step[1190] : Job[11] Step End
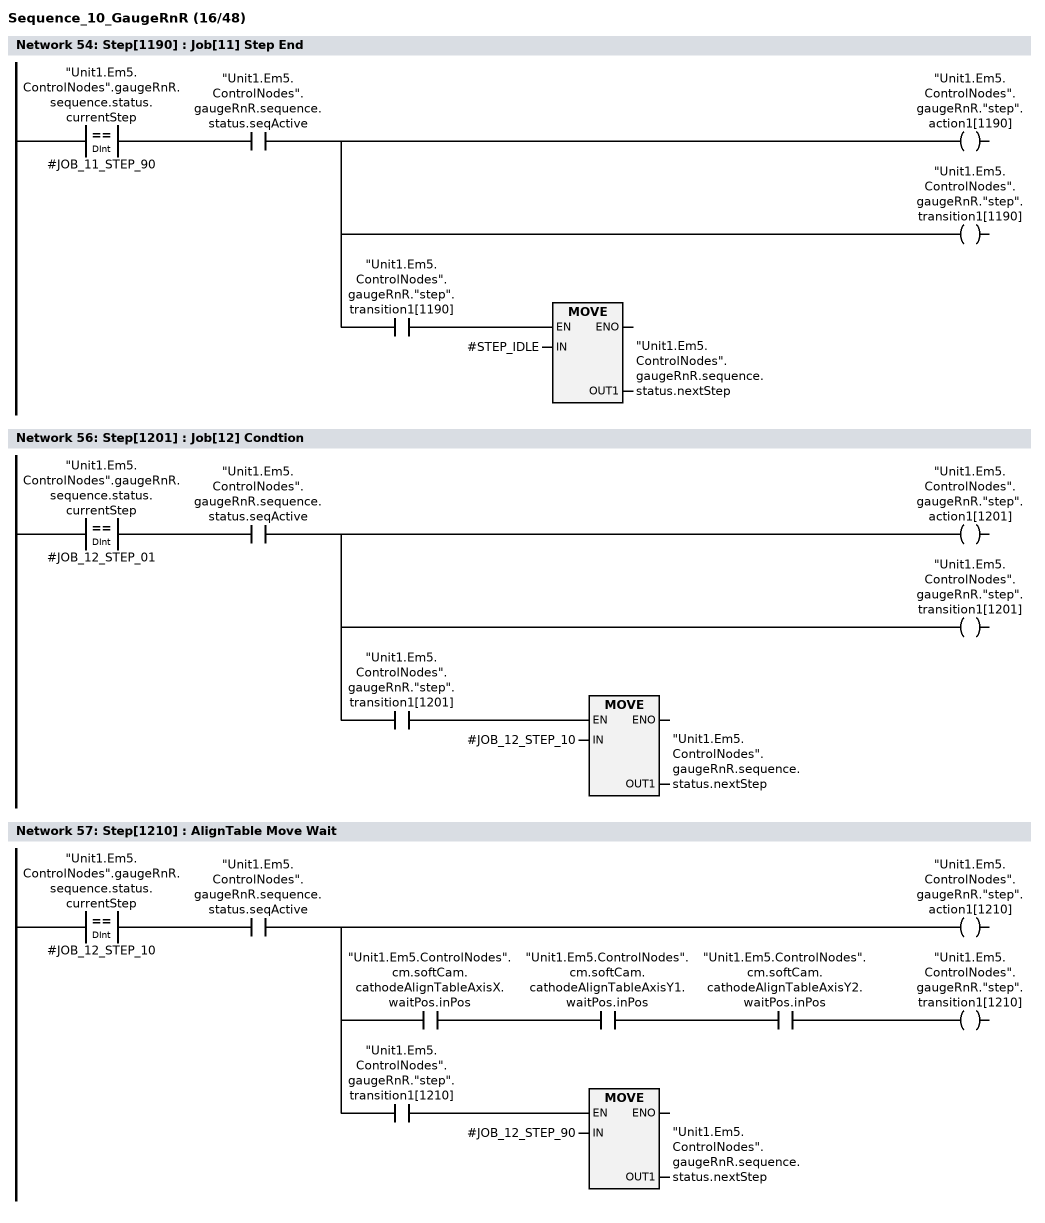
   RUNG wire#powerrail
      { S7_Templates := "SrcType := DInt" } EQ_Contact(in1 := "Unit1.Em5.ControlNodes".gaugeRnR.sequence.status.currentStep, in2 := #JOB_11_STEP_90)
      Contact( "Unit1.Em5.ControlNodes".gaugeRnR.sequence.status.seqActive )
      wire#w1
      Coil( "Unit1.Em5.ControlNodes".gaugeRnR."step".action1[1190] )
   END_RUNG
   RUNG wire#w1
      Coil( "Unit1.Em5.ControlNodes".gaugeRnR."step".transition1[1190] )
   END_RUNG
   RUNG wire#w1
      Contact( "Unit1.Em5.ControlNodes".gaugeRnR."step".transition1[1190] )
      Move(in := #STEP_IDLE, out1 => "Unit1.Em5.ControlNodes".gaugeRnR.sequence.status.nextStep)
   END_RUNG
   // the same network as SCL:
   "Unit1.Em5.ControlNodes".gaugeRnR."step".action1[1190] := ("Unit1.Em5.ControlNodes".gaugeRnR.sequence.status.currentStep = #JOB_11_STEP_90) AND "Unit1.Em5.ControlNodes".gaugeRnR.sequence.status.seqActive;
   "Unit1.Em5.ControlNodes".gaugeRnR."step".transition1[1190] := ("Unit1.Em5.ControlNodes".gaugeRnR.sequence.status.currentStep = #JOB_11_STEP_90) AND "Unit1.Em5.ControlNodes".gaugeRnR.sequence.status.seqActive;
   IF ("Unit1.Em5.ControlNodes".gaugeRnR.sequence.status.currentStep = #JOB_11_STEP_90) AND "Unit1.Em5.ControlNodes".gaugeRnR.sequence.status.seqActive AND "Unit1.Em5.ControlNodes".gaugeRnR."step".transition1[1190] THEN
       "Unit1.Em5.ControlNodes".gaugeRnR.sequence.status.nextStep := #STEP_IDLE;
   END_IF;
END_REGION

REGION Network 55: *************** JOB[12] AlignTable Move Wait ************************
END_REGION

REGION Network 56: Step[1201] : Job[12] Condtion
   RUNG wire#powerrail
      { S7_Templates := "SrcType := DInt" } EQ_Contact(in1 := "Unit1.Em5.ControlNodes".gaugeRnR.sequence.status.currentStep, in2 := #JOB_12_STEP_01)
      Contact( "Unit1.Em5.ControlNodes".gaugeRnR.sequence.status.seqActive )
      wire#w1
      Coil( "Unit1.Em5.ControlNodes".gaugeRnR."step".action1[1201] )
   END_RUNG
   RUNG wire#w1
      Coil( "Unit1.Em5.ControlNodes".gaugeRnR."step".transition1[1201] )
   END_RUNG
   RUNG wire#w1
      Contact( "Unit1.Em5.ControlNodes".gaugeRnR."step".transition1[1201] )
      Move(in := #JOB_12_STEP_10, out1 => "Unit1.Em5.ControlNodes".gaugeRnR.sequence.status.nextStep)
   END_RUNG
   // the same network as SCL:
   "Unit1.Em5.ControlNodes".gaugeRnR."step".action1[1201] := ("Unit1.Em5.ControlNodes".gaugeRnR.sequence.status.currentStep = #JOB_12_STEP_01) AND "Unit1.Em5.ControlNodes".gaugeRnR.sequence.status.seqActive;
   "Unit1.Em5.ControlNodes".gaugeRnR."step".transition1[1201] := ("Unit1.Em5.ControlNodes".gaugeRnR.sequence.status.currentStep = #JOB_12_STEP_01) AND "Unit1.Em5.ControlNodes".gaugeRnR.sequence.status.seqActive;
   IF ("Unit1.Em5.ControlNodes".gaugeRnR.sequence.status.currentStep = #JOB_12_STEP_01) AND "Unit1.Em5.ControlNodes".gaugeRnR.sequence.status.seqActive AND "Unit1.Em5.ControlNodes".gaugeRnR."step".transition1[1201] THEN
       "Unit1.Em5.ControlNodes".gaugeRnR.sequence.status.nextStep := #JOB_12_STEP_10;
   END_IF;
END_REGION

REGION Network 57: Step[1210] : AlignTable Move Wait
   RUNG wire#powerrail
      { S7_Templates := "SrcType := DInt" } EQ_Contact(in1 := "Unit1.Em5.ControlNodes".gaugeRnR.sequence.status.currentStep, in2 := #JOB_12_STEP_10)
      Contact( "Unit1.Em5.ControlNodes".gaugeRnR.sequence.status.seqActive )
      wire#w1
      Coil( "Unit1.Em5.ControlNodes".gaugeRnR."step".action1[1210] )
   END_RUNG
   RUNG wire#w1
      Contact( "Unit1.Em5.ControlNodes".cm.softCam.cathodeAlignTableAxisX.waitPos.inPos )
      Contact( "Unit1.Em5.ControlNodes".cm.softCam.cathodeAlignTableAxisY1.waitPos.inPos )
      Contact( "Unit1.Em5.ControlNodes".cm.softCam.cathodeAlignTableAxisY2.waitPos.inPos )
      Coil( "Unit1.Em5.ControlNodes".gaugeRnR."step".transition1[1210] )
   END_RUNG
   RUNG wire#w1
      Contact( "Unit1.Em5.ControlNodes".gaugeRnR."step".transition1[1210] )
      Move(in := #JOB_12_STEP_90, out1 => "Unit1.Em5.ControlNodes".gaugeRnR.sequence.status.nextStep)
   END_RUNG
   // the same network as SCL:
   "Unit1.Em5.ControlNodes".gaugeRnR."step".action1[1210] := ("Unit1.Em5.ControlNodes".gaugeRnR.sequence.status.currentStep = #JOB_12_STEP_10) AND "Unit1.Em5.ControlNodes".gaugeRnR.sequence.status.seqActive;
   "Unit1.Em5.ControlNodes".gaugeRnR."step".transition1[1210] := ("Unit1.Em5.ControlNodes".gaugeRnR.sequence.status.currentStep = #JOB_12_STEP_10) AND "Unit1.Em5.ControlNodes".gaugeRnR.sequence.status.seqActive AND "Unit1.Em5.ControlNodes".cm.softCam.cathodeAlignTableAxisX.waitPos.inPos AND "Unit1.Em5.ControlNodes".cm.softCam.cathodeAlignTableAxisY1.waitPos.inPos AND "Unit1.Em5.ControlNodes".cm.softCam.cathodeAlignTableAxisY2.waitPos.inPos;
   IF ("Unit1.Em5.ControlNodes".gaugeRnR.sequence.status.currentStep = #JOB_12_STEP_10) AND "Unit1.Em5.ControlNodes".gaugeRnR.sequence.status.seqActive AND "Unit1.Em5.ControlNodes".gaugeRnR."step".transition1[1210] THEN
       "Unit1.Em5.ControlNodes".gaugeRnR.sequence.status.nextStep := #JOB_12_STEP_90;
   END_IF;
END_REGION

REGION Network 58: Step[1290] : Job[12] Step End
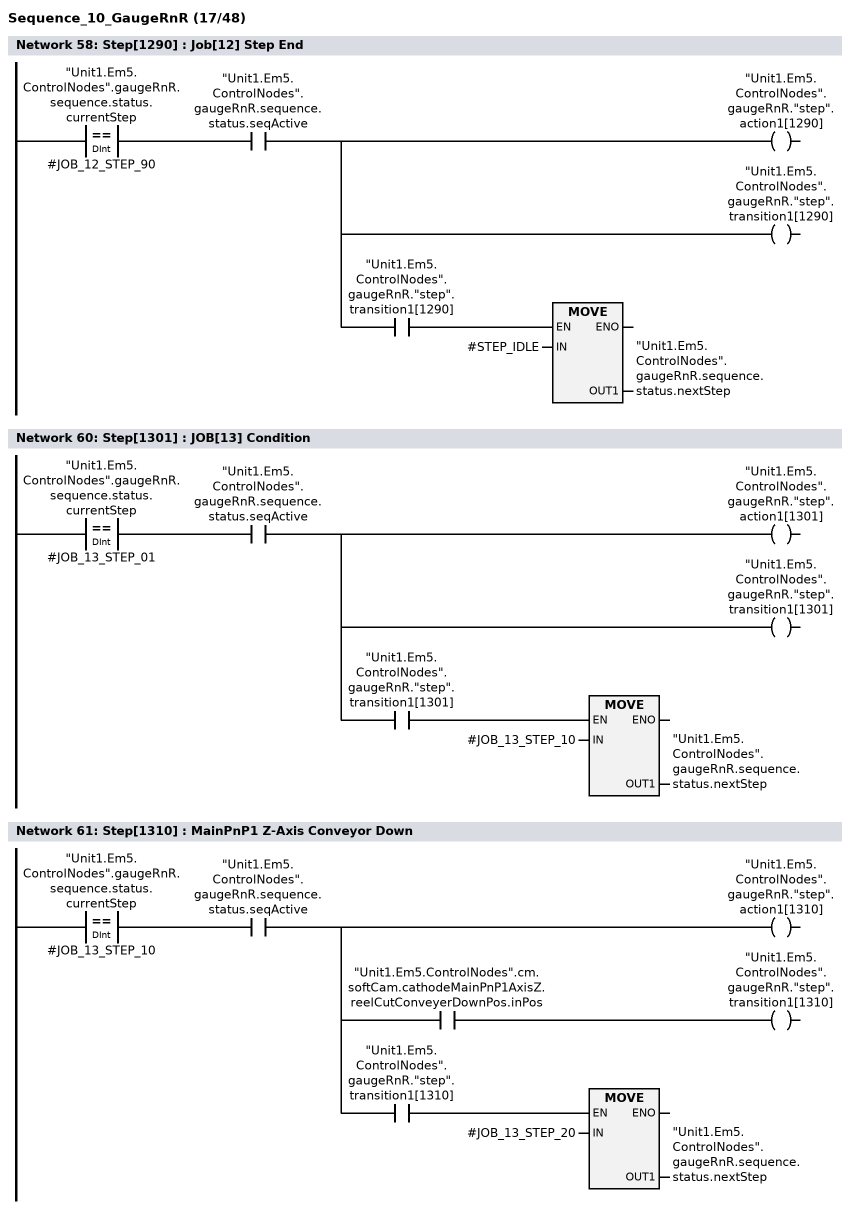
   RUNG wire#powerrail
      { S7_Templates := "SrcType := DInt" } EQ_Contact(in1 := "Unit1.Em5.ControlNodes".gaugeRnR.sequence.status.currentStep, in2 := #JOB_12_STEP_90)
      Contact( "Unit1.Em5.ControlNodes".gaugeRnR.sequence.status.seqActive )
      wire#w1
      Coil( "Unit1.Em5.ControlNodes".gaugeRnR."step".action1[1290] )
   END_RUNG
   RUNG wire#w1
      Coil( "Unit1.Em5.ControlNodes".gaugeRnR."step".transition1[1290] )
   END_RUNG
   RUNG wire#w1
      Contact( "Unit1.Em5.ControlNodes".gaugeRnR."step".transition1[1290] )
      Move(in := #STEP_IDLE, out1 => "Unit1.Em5.ControlNodes".gaugeRnR.sequence.status.nextStep)
   END_RUNG
   // the same network as SCL:
   "Unit1.Em5.ControlNodes".gaugeRnR."step".action1[1290] := ("Unit1.Em5.ControlNodes".gaugeRnR.sequence.status.currentStep = #JOB_12_STEP_90) AND "Unit1.Em5.ControlNodes".gaugeRnR.sequence.status.seqActive;
   "Unit1.Em5.ControlNodes".gaugeRnR."step".transition1[1290] := ("Unit1.Em5.ControlNodes".gaugeRnR.sequence.status.currentStep = #JOB_12_STEP_90) AND "Unit1.Em5.ControlNodes".gaugeRnR.sequence.status.seqActive;
   IF ("Unit1.Em5.ControlNodes".gaugeRnR.sequence.status.currentStep = #JOB_12_STEP_90) AND "Unit1.Em5.ControlNodes".gaugeRnR.sequence.status.seqActive AND "Unit1.Em5.ControlNodes".gaugeRnR."step".transition1[1290] THEN
       "Unit1.Em5.ControlNodes".gaugeRnR.sequence.status.nextStep := #STEP_IDLE;
   END_IF;
END_REGION

REGION Network 59: *************** JOB[13] Unload MasterPiece ************************
END_REGION

REGION Network 60: Step[1301] : JOB[13] Condition
   RUNG wire#powerrail
      { S7_Templates := "SrcType := DInt" } EQ_Contact(in1 := "Unit1.Em5.ControlNodes".gaugeRnR.sequence.status.currentStep, in2 := #JOB_13_STEP_01)
      Contact( "Unit1.Em5.ControlNodes".gaugeRnR.sequence.status.seqActive )
      wire#w1
      Coil( "Unit1.Em5.ControlNodes".gaugeRnR."step".action1[1301] )
   END_RUNG
   RUNG wire#w1
      Coil( "Unit1.Em5.ControlNodes".gaugeRnR."step".transition1[1301] )
   END_RUNG
   RUNG wire#w1
      Contact( "Unit1.Em5.ControlNodes".gaugeRnR."step".transition1[1301] )
      Move(in := #JOB_13_STEP_10, out1 => "Unit1.Em5.ControlNodes".gaugeRnR.sequence.status.nextStep)
   END_RUNG
   // the same network as SCL:
   "Unit1.Em5.ControlNodes".gaugeRnR."step".action1[1301] := ("Unit1.Em5.ControlNodes".gaugeRnR.sequence.status.currentStep = #JOB_13_STEP_01) AND "Unit1.Em5.ControlNodes".gaugeRnR.sequence.status.seqActive;
   "Unit1.Em5.ControlNodes".gaugeRnR."step".transition1[1301] := ("Unit1.Em5.ControlNodes".gaugeRnR.sequence.status.currentStep = #JOB_13_STEP_01) AND "Unit1.Em5.ControlNodes".gaugeRnR.sequence.status.seqActive;
   IF ("Unit1.Em5.ControlNodes".gaugeRnR.sequence.status.currentStep = #JOB_13_STEP_01) AND "Unit1.Em5.ControlNodes".gaugeRnR.sequence.status.seqActive AND "Unit1.Em5.ControlNodes".gaugeRnR."step".transition1[1301] THEN
       "Unit1.Em5.ControlNodes".gaugeRnR.sequence.status.nextStep := #JOB_13_STEP_10;
   END_IF;
END_REGION

REGION Network 61: Step[1310] : MainPnP1 Z-Axis Conveyor Down
   RUNG wire#powerrail
      { S7_Templates := "SrcType := DInt" } EQ_Contact(in1 := "Unit1.Em5.ControlNodes".gaugeRnR.sequence.status.currentStep, in2 := #JOB_13_STEP_10)
      Contact( "Unit1.Em5.ControlNodes".gaugeRnR.sequence.status.seqActive )
      wire#w1
      Coil( "Unit1.Em5.ControlNodes".gaugeRnR."step".action1[1310] )
   END_RUNG
   RUNG wire#w1
      Contact( "Unit1.Em5.ControlNodes".cm.softCam.cathodeMainPnP1AxisZ.reelCutConveyerDownPos.inPos )
      Coil( "Unit1.Em5.ControlNodes".gaugeRnR."step".transition1[1310] )
   END_RUNG
   RUNG wire#w1
      Contact( "Unit1.Em5.ControlNodes".gaugeRnR."step".transition1[1310] )
      Move(in := #JOB_13_STEP_20, out1 => "Unit1.Em5.ControlNodes".gaugeRnR.sequence.status.nextStep)
   END_RUNG
   // the same network as SCL:
   "Unit1.Em5.ControlNodes".gaugeRnR."step".action1[1310] := ("Unit1.Em5.ControlNodes".gaugeRnR.sequence.status.currentStep = #JOB_13_STEP_10) AND "Unit1.Em5.ControlNodes".gaugeRnR.sequence.status.seqActive;
   "Unit1.Em5.ControlNodes".gaugeRnR."step".transition1[1310] := ("Unit1.Em5.ControlNodes".gaugeRnR.sequence.status.currentStep = #JOB_13_STEP_10) AND "Unit1.Em5.ControlNodes".gaugeRnR.sequence.status.seqActive AND "Unit1.Em5.ControlNodes".cm.softCam.cathodeMainPnP1AxisZ.reelCutConveyerDownPos.inPos;
   IF ("Unit1.Em5.ControlNodes".gaugeRnR.sequence.status.currentStep = #JOB_13_STEP_10) AND "Unit1.Em5.ControlNodes".gaugeRnR.sequence.status.seqActive AND "Unit1.Em5.ControlNodes".gaugeRnR."step".transition1[1310] THEN
       "Unit1.Em5.ControlNodes".gaugeRnR.sequence.status.nextStep := #JOB_13_STEP_20;
   END_IF;
END_REGION

REGION Network 62: Step[1320] : MainPnP1 Vaccum Off
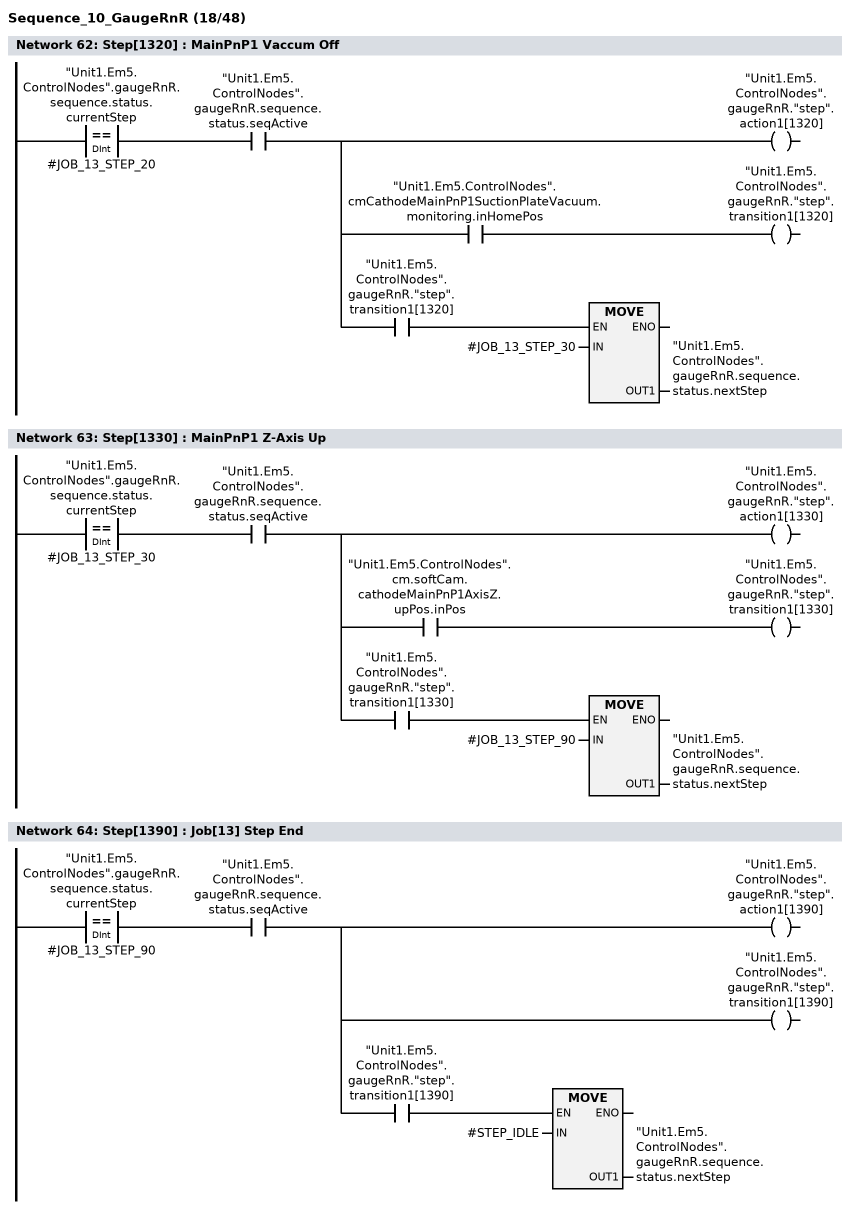
   RUNG wire#powerrail
      { S7_Templates := "SrcType := DInt" } EQ_Contact(in1 := "Unit1.Em5.ControlNodes".gaugeRnR.sequence.status.currentStep, in2 := #JOB_13_STEP_20)
      Contact( "Unit1.Em5.ControlNodes".gaugeRnR.sequence.status.seqActive )
      wire#w1
      Coil( "Unit1.Em5.ControlNodes".gaugeRnR."step".action1[1320] )
   END_RUNG
   RUNG wire#w1
      Contact( "Unit1.Em5.ControlNodes".cmCathodeMainPnP1SuctionPlateVacuum.monitoring.inHomePos )
      Coil( "Unit1.Em5.ControlNodes".gaugeRnR."step".transition1[1320] )
   END_RUNG
   RUNG wire#w1
      Contact( "Unit1.Em5.ControlNodes".gaugeRnR."step".transition1[1320] )
      Move(in := #JOB_13_STEP_30, out1 => "Unit1.Em5.ControlNodes".gaugeRnR.sequence.status.nextStep)
   END_RUNG
   // the same network as SCL:
   "Unit1.Em5.ControlNodes".gaugeRnR."step".action1[1320] := ("Unit1.Em5.ControlNodes".gaugeRnR.sequence.status.currentStep = #JOB_13_STEP_20) AND "Unit1.Em5.ControlNodes".gaugeRnR.sequence.status.seqActive;
   "Unit1.Em5.ControlNodes".gaugeRnR."step".transition1[1320] := ("Unit1.Em5.ControlNodes".gaugeRnR.sequence.status.currentStep = #JOB_13_STEP_20) AND "Unit1.Em5.ControlNodes".gaugeRnR.sequence.status.seqActive AND "Unit1.Em5.ControlNodes".cmCathodeMainPnP1SuctionPlateVacuum.monitoring.inHomePos;
   IF ("Unit1.Em5.ControlNodes".gaugeRnR.sequence.status.currentStep = #JOB_13_STEP_20) AND "Unit1.Em5.ControlNodes".gaugeRnR.sequence.status.seqActive AND "Unit1.Em5.ControlNodes".gaugeRnR."step".transition1[1320] THEN
       "Unit1.Em5.ControlNodes".gaugeRnR.sequence.status.nextStep := #JOB_13_STEP_30;
   END_IF;
END_REGION

REGION Network 63: Step[1330] : MainPnP1 Z-Axis Up
   RUNG wire#powerrail
      { S7_Templates := "SrcType := DInt" } EQ_Contact(in1 := "Unit1.Em5.ControlNodes".gaugeRnR.sequence.status.currentStep, in2 := #JOB_13_STEP_30)
      Contact( "Unit1.Em5.ControlNodes".gaugeRnR.sequence.status.seqActive )
      wire#w1
      Coil( "Unit1.Em5.ControlNodes".gaugeRnR."step".action1[1330] )
   END_RUNG
   RUNG wire#w1
      Contact( "Unit1.Em5.ControlNodes".cm.softCam.cathodeMainPnP1AxisZ.upPos.inPos )
      Coil( "Unit1.Em5.ControlNodes".gaugeRnR."step".transition1[1330] )
   END_RUNG
   RUNG wire#w1
      Contact( "Unit1.Em5.ControlNodes".gaugeRnR."step".transition1[1330] )
      Move(in := #JOB_13_STEP_90, out1 => "Unit1.Em5.ControlNodes".gaugeRnR.sequence.status.nextStep)
   END_RUNG
   // the same network as SCL:
   "Unit1.Em5.ControlNodes".gaugeRnR."step".action1[1330] := ("Unit1.Em5.ControlNodes".gaugeRnR.sequence.status.currentStep = #JOB_13_STEP_30) AND "Unit1.Em5.ControlNodes".gaugeRnR.sequence.status.seqActive;
   "Unit1.Em5.ControlNodes".gaugeRnR."step".transition1[1330] := ("Unit1.Em5.ControlNodes".gaugeRnR.sequence.status.currentStep = #JOB_13_STEP_30) AND "Unit1.Em5.ControlNodes".gaugeRnR.sequence.status.seqActive AND "Unit1.Em5.ControlNodes".cm.softCam.cathodeMainPnP1AxisZ.upPos.inPos;
   IF ("Unit1.Em5.ControlNodes".gaugeRnR.sequence.status.currentStep = #JOB_13_STEP_30) AND "Unit1.Em5.ControlNodes".gaugeRnR.sequence.status.seqActive AND "Unit1.Em5.ControlNodes".gaugeRnR."step".transition1[1330] THEN
       "Unit1.Em5.ControlNodes".gaugeRnR.sequence.status.nextStep := #JOB_13_STEP_90;
   END_IF;
END_REGION

